	PLC_RECV1.m_nExpId 			:=  PLC_RECV1.m_nExpId 			;      
	PLC_RECV1.m_nAngleStart 	:=	PLC_RECV1.m_nAngleStart 	;   
	PLC_RECV1.m_nAngleEnd  		:=	PLC_RECV1.m_nAngleEnd  		;   
	PLC_RECV1.m_nRotateBegin  	:=  PLC_RECV1.m_nRotateBegin  	; 
	PLC_RECV1.m_nRotateEnd  	:=	PLC_RECV1.m_nRotateEnd  	;   
	PLC_RECV1.m_nKv  			:=	PLC_RECV1.m_nKv  			;       
	PLC_RECV1.m_nMA  			:=	PLC_RECV1.m_nMA  			;        
	PLC_RECV1.m_nMS 			:=	PLC_RECV1.m_nMS 			;        
	PLC_RECV1.m_nFocus 			:=  PLC_RECV1.m_nFocus 			;     
	PLC_RECV1.m_nAcquireFrame 	:=  PLC_RECV1.m_nAcquireFrame 	;
	PLC_RECV1.m_nFramePerCirCle	:=  PLC_RECV1.m_nFramePerCirCle	;
	PLC_RECV1.m_nMoveToward  	:=	PLC_RECV1.m_nMoveToward  	 ;
	PLC_RECV1.m_nServenLamp  	:=  PLC_RECV1.m_nServenLamp  	 ;
	PLC_RECV1.m_nMoveStep  		:=  PLC_RECV1.m_nMoveStep  		 ;  
	PLC_RECV1.m_nPitchValue   	:=  PLC_RECV1.m_nPitchValue   	 ;
	PLC_RECV1.m_nCircleCount  	:=  PLC_RECV1.m_nCircleCount  	 ;
	PLC_RECV1.m_nControlState 	:=  PLC_RECV1.m_nControlState 	 ;
	PLC_RECV1.m_fScanTop 		:=	PLC_RECV1.m_fScanTop 		 ;    
	PLC_RECV1.m_fScanBottom 	:=	PLC_RECV1.m_fScanBottom 	 ;  
	PLC_RECV1.m_fSecondPerCicle	:=  PLC_RECV1.m_fSecondPerCicle	;
	PLC_RECV1.m_nSamplingRate  	:=  PLC_RECV1.m_nSamplingRate  	;
	PLC_RECV1.m_nPrepareState 	:=  PLC_RECV1.m_nPrepareState 	 ;
	PLC_RECV1.m_nScanMoveType	:=	PLC_RECV1.m_nScanMoveType	;  
	PLC_RECV1.m_nCircleIndex 	:=	PLC_RECV1.m_nCircleIndex 	;  
	PLC_RECV1.m_nPLCMaCoeff 	:=	PLC_RECV1.m_nPLCMaCoeff 	 ;  
	PLC_RECV1.m_nLastMsg  		:=  PLC_RECV1.m_nLastMsg  		;    
	PLC_RECV1.m_nDelayTime 		:=  PLC_RECV1.m_nDelayTime 		;       
	PLC_RECV1.yuliu_2			:=	PLC_RECV1.yuliu_2			 ;       
	PLC_RECV1.yuliu_3 			:=  PLC_RECV1.yuliu_3 			 ;      	
END_IF
END_ACTION

ACTION APLC_SENG:

(*---------------------------------PLC发送数据------------------------------------*)//大端发送机制
(*第一部分，发送数据赋值,待补充*)
	IF PLC_RECV1.m_nSocketType=1 THEN
    	PLC_SEND1.m_nSocketType	  := 1;//心跳指令，默认为3，留待判断连接状态。
	ELSE
    	PLC_SEND1.m_nSocketType	  := 3;//心跳指令，默认为3，留待判断连接状态。
	END_IF                                                                            
	PLC_SEND1.m_nCurrentAngle	:= LREAL_TO_REAL(Axis_XZ.XZ_AxisState.rActPosition);//为设备当前的旋转角度，单位为角度制下的单位，为度。数精度为1度；                                                             
	PLC_SEND1.m_nBedHeight		:= Entity_IO.rRealPos+710; //为床高，单位为毫米，数据范围为0 - 2000mm；                                                                 
	PLC_SEND1.m_nBedMovePos		:= LREAL_TO_REAL(Axis_QJ.QJ_AxisState.rActPosition);//为床移动距离，以床与探测板的垂直面交线为起点，单位为毫米，数据范围为0 - 3000mm；//增加了偏移                                                 
//	PLC_SEND1.m_nExpStates		:= 22;//为曝光状态，枚举值，0:idle（空闲） 1:prep（训机） 2: ready（训机结束，准备完成，可以出束） 3: XrayOn（出射线） 4:XrayOff（关射线） 5 error；
	PLC_SEND1.m_nExpCount		:= PLC_PRG.iActNumPulse;//为曝光的次数，对应曝光的图像张数；                                                                              
//	PLC_SEND1.m_nFocus			:= XRAY_RS485.Feedback_nFocus;//焦点大小，0为大焦点 1为小焦点， 焦点具体对应的值由plc设置；        //修改为按键提示                                                      
	PLC_SEND1.m_nMHuValue		:= DT_Xray.Feedback_nMHuValue;//热容量，单位MHu ，实际热容量*100得到，实际热容量为小数；                                                               
	PLC_SEND1.m_nDirectionState	:= BOOL_TO_UDINT(PLC_PRG.bSendQuickCTAngle);                                                                  
//	PLC_SEND1.m_nMoveState		:= 22;//起始、终止状态， 默认值-1， 0为当前扫描方案（与常规意义不同，注意区别）处于准备好状态，可以准备扫描；1为当前扫描方案结束，运动过程中值为-1                      
	PLC_SEND1.m_nError			:= DT_Xray.iAlarmNum;//错误码使用，由王（风杰）工具体阐述内容                                                                            
	PLC_SEND1.m_fSpeed			:= LREAL_TO_REAL(Axis_XZ.XZ_AxisState.rActVelocity);//为设备的旋转速度，单位为度/秒，精度0.01度/秒；                                                                     
	PLC_SEND1.m_fKv				:= DT_Xray.Feedback_Kv;//管电压，单位为kv（千伏），精度0.01；                                                                          
	PLC_SEND1.m_fMA				:= DT_Xray.Feedback_mA;//管电流，单位为mA（毫安），精度0.01；                                                                          
	PLC_SEND1.m_fMs				:= DT_Xray.Feedback_ms;//曝光时间，单位为ms（毫秒），精度0.01；                                                                         
	PLC_SEND1.m_nSamplingRate	:= PLC_RECV1.m_nFramePerCirCle;//采样率，有3个选项：2400帧/圈；1200帧/圈；600帧/圈                                                               
//	PLC_SEND1.m_nScanProType	:= 22;//执行扫描方案的类型，0为自动扫描，1为手动扫描，2为无设置意义的值，默认值为2                                                        
	PLC_SEND1.PLC_State			:= GVL_State.iPLC_State;//PLC状态机状态                                                                                             
	PLC_SEND1.XRAY_State		:= GVL_State.iXray_State;//射线源状态                                                                                     
	PLC_SEND1.AxisErrorID		:= QJ_Error+XZ_Error*65536; //电机错误报警位,各占16位 
    PLC_SEND1.m_nFocusX			:= DT_Xray.Feedback_nFocus;//反馈的焦点

(**处理电机Errstop状态下没有故障吗的情况*)	
	IF Axis_XZ.XZ_AxisState.bAxisErr THEN
		XZ_Error:= Axis_XZ.XZ_AxisState.ErrorID ;
	ELSE
		IF  Axis_XZ.XZ_AxisState.bErrStop THEN
			XZ_Error:= 444 ; 
		ELSE
			XZ_Error:=0;
		END_IF
	END_IF
	
	IF Axis_QJ.QJ_AxisState.bAxisErr THEN
		XZ_Error:= Axis_QJ.QJ_AxisState.ErrorID ;
	ELSE
		IF  Axis_QJ.QJ_AxisState.bErrStop THEN
			QJ_Error:= 444 ; 
		ELSE
			QJ_Error:=0;
		END_IF
	END_IF
	                               
(*第二部分，发送数据发送*)
(*1,//心跳指令，默认为3，留待判断连接状态。*)
	abyWriteData[3]:=UDINT_TO_BYTE(ROR((PLC_SEND1.m_nSocketType AND 16#FF000000),24));
	abyWriteData[2]:=UDINT_TO_BYTE(ROR((PLC_SEND1.m_nSocketType AND 16#FF0000),16));
	abyWriteData[1]:=UDINT_TO_BYTE(ROR((PLC_SEND1.m_nSocketType AND 16#FF00),8));
	abyWriteData[0]:=UDINT_TO_BYTE(PLC_SEND1.m_nSocketType);
	
(*2//为设备当前的旋转角度，单位为角度制下的单位，为度，数精度为1度*)
	RealByte1[0].rData:=PLC_SEND1.m_nCurrentAngle;	
	abyWriteData[4]:=RealByte1[0].wByte[0];
	abyWriteData[5]:=RealByte1[0].wByte[1];
	abyWriteData[6]:=RealByte1[0].wByte[2];
	abyWriteData[7]:=RealByte1[0].wByte[3];
	
(*3//为床高，单位为毫米，数据范围为0 - 2000mm；*)
	RealByte1[1].rData:=PLC_SEND1.m_nBedHeight;	
	abyWriteData[8]:=RealByte1[1].wByte[0];
	abyWriteData[9]:=RealByte1[1].wByte[1];
	abyWriteData[10]:=RealByte1[1].wByte[2];
	abyWriteData[11]:=RealByte1[1].wByte[3];
	
(*4//为床移动距离，以床与探测板的垂直面交线为起点，单位为毫米，数据范围为0 - 3000mm；*)
	RealByte1[2].rData:=PLC_SEND1.m_nBedMovePos;	
	abyWriteData[12]:=RealByte1[2].wByte[0];
	abyWriteData[13]:=RealByte1[2].wByte[1];
	abyWriteData[14]:=RealByte1[2].wByte[2];
	abyWriteData[15]:=RealByte1[2].wByte[3];
	
(*5//为曝光状态，枚举值，0:idle（空闲） 1:prep（训机） 2: ready（训机结束，准备完成，可以出束） 3: XrayOn（出射线） 4:XrayOff（关射线） 5 error；*)
	abyWriteData[19]:=UDINT_TO_BYTE(ROR((PLC_SEND1.m_nExpStates AND 16#FF000000),24));
	abyWriteData[18]:=UDINT_TO_BYTE(ROR((PLC_SEND1.m_nExpStates AND 16#FF0000),16));
	abyWriteData[17]:=UDINT_TO_BYTE(ROR((PLC_SEND1.m_nExpStates AND 16#FF00),8));
	abyWriteData[16]:=UDINT_TO_BYTE(PLC_SEND1.m_nExpStates);
	
(*6//为曝光的次数，对应曝光的图像张数*)
	abyWriteData[23]:=UDINT_TO_BYTE(ROR((PLC_SEND1.m_nExpCount AND 16#FF000000),24));
	abyWriteData[22]:=UDINT_TO_BYTE(ROR((PLC_SEND1.m_nExpCount AND 16#FF0000),16));
	abyWriteData[21]:=UDINT_TO_BYTE(ROR((PLC_SEND1.m_nExpCount AND 16#FF00),8));
	abyWriteData[20]:=UDINT_TO_BYTE(PLC_SEND1.m_nExpCount AND 16#FF);
	
(*7//焦点大小，0为大焦点 1为小焦点， 焦点具体对应的值由plc设置；*)
	abyWriteData[27]:=UDINT_TO_BYTE(ROR((PLC_SEND1.m_nFocus AND 16#FF000000),24));
	abyWriteData[26]:=UDINT_TO_BYTE(ROR((PLC_SEND1.m_nFocus AND 16#FF0000),16));
	abyWriteData[25]:=UDINT_TO_BYTE(ROR((PLC_SEND1.m_nFocus AND 16#FF00),8));
	abyWriteData[24]:=UDINT_TO_BYTE(PLC_SEND1.m_nFocus);

(*8////热容量，单位MHu ，实际热容量*100得到，实际热容量为小数；*)
	RealByte1[3].rData:=PLC_SEND1.m_nMHuValue;	
	abyWriteData[28]:=RealByte1[3].wByte[0];
	abyWriteData[29]:=RealByte1[3].wByte[1];
	abyWriteData[30]:=RealByte1[3].wByte[2];
	abyWriteData[31]:=RealByte1[3].wByte[3];

(*9.;//当前旋转状态，默认值0， 1为正转，2为反转，停止为0*)	
	abyWriteData[35]:=UDINT_TO_BYTE(ROR((PLC_SEND1.m_nDirectionState AND 16#FF000000),24));
	abyWriteData[34]:=UDINT_TO_BYTE(ROR((PLC_SEND1.m_nDirectionState AND 16#FF0000),16));
	abyWriteData[33]:=UDINT_TO_BYTE(ROR((PLC_SEND1.m_nDirectionState AND 16#FF00),8));
	abyWriteData[32]:=UDINT_TO_BYTE(PLC_SEND1.m_nDirectionState);
	
(*10.起始、终止状态， 默认值0， 1为当前扫描方案（与常规意义不同，注意区别）处于准备好状态，可以准备扫描；2为当前扫描方案结束，运动过程中值为0*)
	abyWriteData[39]:=UDINT_TO_BYTE(ROR((PLC_SEND1.m_nMoveState AND 16#FF000000),24));
	abyWriteData[38]:=UDINT_TO_BYTE(ROR((PLC_SEND1.m_nMoveState AND 16#FF0000),16));
	abyWriteData[37]:=UDINT_TO_BYTE(ROR((PLC_SEND1.m_nMoveState AND 16#FF00),8));
	abyWriteData[36]:=UDINT_TO_BYTE(PLC_SEND1.m_nMoveState);
	
(*11.//错误码使用*)
	abyWriteData[43]:=UDINT_TO_BYTE(ROR((PLC_SEND1.m_nError AND 16#FF000000),24));
	abyWriteData[42]:=UDINT_TO_BYTE(ROR((PLC_SEND1.m_nError AND 16#FF0000),16));
	abyWriteData[41]:=UDINT_TO_BYTE(ROR((PLC_SEND1.m_nError AND 16#FF00),8));
	abyWriteData[40]:=UDINT_TO_BYTE(PLC_SEND1.m_nError AND 16#FF);//旋转电机错误码
	
(*12.//为设备的旋转速度，单位为度/秒，精度0.01度/秒；*)
	RealByte1[4].rData:=PLC_SEND1.m_fSpeed;	
	abyWriteData[44]:=RealByte1[4].wByte[0];
	abyWriteData[45]:=RealByte1[4].wByte[1];
	abyWriteData[46]:=RealByte1[4].wByte[2];
	abyWriteData[47]:=RealByte1[4].wByte[3];
	
(*13.//管电压，单位为kv（千伏），精度1；*)
	abyWriteData[51]:=UDINT_TO_BYTE(ROR((PLC_SEND1.m_fKv AND 16#FF000000),24));
	abyWriteData[50]:=UDINT_TO_BYTE(ROR((PLC_SEND1.m_fKv AND 16#FF0000),16));
	abyWriteData[49]:=UDINT_TO_BYTE(ROR((PLC_SEND1.m_fKv AND 16#FF00),8));
	abyWriteData[48]:=UDINT_TO_BYTE(PLC_SEND1.m_fKv AND 16#FF);
	
(*14.//管电流，单位为mA（毫安），精度0.1*)
	RealByte1[6].rData:=PLC_SEND1.m_fMA;	
	abyWriteData[52]:=RealByte1[6].wByte[0];
	abyWriteData[53]:=RealByte1[6].wByte[1];
	abyWriteData[54]:=RealByte1[6].wByte[2];
	abyWriteData[55]:=RealByte1[6].wByte[3];

(*15.//曝光时间，单位为ms（毫秒），精度0.01；*)
	RealByte1[7].rData:=PLC_SEND1.m_fMs;	
	abyWriteData[56]:=RealByte1[7].wByte[0];
	abyWriteData[57]:=RealByte1[7].wByte[1];
	abyWriteData[58]:=RealByte1[7].wByte[2];
	abyWriteData[59]:=RealByte1[7].wByte[3];
	
(*16.//采样率，有3个选项：2400帧/圈；1200帧/圈；600帧/圈*)
	abyWriteData[63]:=UDINT_TO_BYTE(ROR((PLC_SEND1.m_nSamplingRate AND 16#FF000000),24));
	abyWriteData[62]:=UDINT_TO_BYTE(ROR((PLC_SEND1.m_nSamplingRate AND 16#FF0000),16));
	abyWriteData[61]:=UDINT_TO_BYTE(ROR((PLC_SEND1.m_nSamplingRate AND 16#FF00),8));
	abyWriteData[60]:=UDINT_TO_BYTE(PLC_SEND1.m_nSamplingRate AND 16#FF);
	
(*17.//执行扫描方案的类型，0为自动扫描，1为手动扫描，2为无设置意义的值，默认值为2*)
	abyWriteData[67]:=UDINT_TO_BYTE(ROR((PLC_SEND1.m_nScanProType AND 16#FF000000),24));
	abyWriteData[66]:=UDINT_TO_BYTE(ROR((PLC_SEND1.m_nScanProType AND 16#FF0000),16));
	abyWriteData[65]:=UDINT_TO_BYTE(ROR((PLC_SEND1.m_nScanProType AND 16#FF00),8));
	abyWriteData[64]:=UDINT_TO_BYTE(PLC_SEND1.m_nScanProType AND 16#FF);
	
(*18.//PLC工作状态*)
	abyWriteData[71]:=UDINT_TO_BYTE(ROR((PLC_SEND1.PLC_State AND 16#FF000000),24));
	abyWriteData[70]:=UDINT_TO_BYTE(ROR((PLC_SEND1.PLC_State AND 16#FF0000),16));//
	abyWriteData[69]:=UDINT_TO_BYTE(ROR((PLC_SEND1.PLC_State AND 16#FF00),8));	///
	abyWriteData[68]:=UDINT_TO_BYTE(PLC_SEND1.PLC_State AND 16#FF);				//PLC状态机
	
(*19.//XRAY状态*)
	abyWriteData[75]:=UDINT_TO_BYTE(ROR((PLC_SEND1.XRAY_State AND 16#FF000000),24));
	abyWriteData[74]:=UDINT_TO_BYTE(ROR((PLC_SEND1.XRAY_State AND 16#FF0000),16));  
	abyWriteData[73]:=UDINT_TO_BYTE(ROR((PLC_SEND1.XRAY_State AND 16#FF00),8));     
	abyWriteData[72]:=UDINT_TO_BYTE(PLC_SEND1.XRAY_State AND 16#FF);  //射线源状态机              
	
(*20.//电机错误码*)
	abyWriteData[79]:=UDINT_TO_BYTE(ROR((PLC_SEND1.AxisErrorID AND 16#FF000000),24));//旋转电机故障码
	abyWriteData[78]:=UDINT_TO_BYTE(ROR((PLC_SEND1.AxisErrorID AND 16#FF0000),16));//旋转电机故障码
	abyWriteData[77]:=UDINT_TO_BYTE(ROR((PLC_SEND1.AxisErrorID AND 16#FF00),8));//前进电机故障码
	abyWriteData[76]:=UDINT_TO_BYTE(PLC_SEND1.AxisErrorID AND 16#FF);//前进电机故障码
	
(*21.射线源大小焦点反馈*)
	abyWriteData[83]:=UDINT_TO_BYTE(ROR((PLC_SEND1.m_nFocusX AND 16#FF000000),24));//
	abyWriteData[82]:=UDINT_TO_BYTE(ROR((PLC_SEND1.m_nFocusX AND 16#FF0000),16));//
	abyWriteData[81]:=UDINT_TO_BYTE(ROR((PLC_SEND1.m_nFocusX AND 16#FF00),8));//
	abyWriteData[80]:=UDINT_TO_BYTE(PLC_SEND1.m_nFocusX AND 16#FF);//反馈焦点
	
	
(*	TEST
	PLC_SEND1.m_nSocketType	  	:= 1;//心跳指令，默认为3，留待判断连接状态。                                                                            
	PLC_SEND1.m_nCurrentAngle	:= 2.1;//为设备当前的旋转角度，单位为角度制下的单位，为度。数精度为1度；                                                               
	PLC_SEND1.m_nBedHeight		:= 3.2;//为床高，单位为毫米，数据范围为0 - 2000mm；                                                                  
	PLC_SEND1.m_nBedMovePos		:= 4.3;//为床移动距离，以床与探测板的垂直面交线为起点，单位为毫米，数据范围为0 - 3000mm；                                                  
	PLC_SEND1.m_nExpStates		:= 5;//为曝光状态，枚举值，0:idle（空闲） 1:prep（训机） 2: ready（训机结束，准备完成，可以出束） 3: XrayOn（出射线） 4:XrayOff（关射线） 5 error；
	PLC_SEND1.m_nExpCount		:= 6;//为曝光的次数，对应曝光的图像张数；                                                                              
	PLC_SEND1.m_nFocus			:= 7;//焦点大小，0为大焦点 1为小焦点， 焦点具体对应的值由plc设置；                                                              
	PLC_SEND1.m_nMHuValue		:= 8.1;//热容量，单位MHu ，实际热容量*100得到，实际热容量为小数；                                                               
	PLC_SEND1.m_nDirectionState	:= 9;//当前旋转状态，默认值-1， 0为正转，1为反转，停止为-1                                                                  
	PLC_SEND1.m_nMoveState		:= 10;//起始、终止状态， 默认值-1， 0为当前扫描方案（与常规意义不同，注意区别）处于准备好状态，可以准备扫描；1为当前扫描方案结束，运动过程中值为-1                      
	PLC_SEND1.m_nError			:= 11;//错误码使用，由王（风杰）工具体阐述内容                                                                            
	PLC_SEND1.m_fSpeed			:= 12.2;//为设备的旋转速度，单位为度/秒，精度0.01度/秒；                                                                     
	PLC_SEND1.m_fKv				:= 13;//管电压，单位为kv（千伏），精度0.01；                                                                          
	PLC_SEND1.m_fMA				:= 14.3;//管电流，单位为mA（毫安），精度0.01；                                                                          
	PLC_SEND1.m_fMs				:= 15.3;//曝光时间，单位为ms（毫秒），精度0.01；                                                                         
	PLC_SEND1.m_nSamplingRate	:= 16;//采样率，有3个选项：2400帧/圈；1200帧/圈；600帧/圈                                                               
	PLC_SEND1.m_nScanProType	:= 17;//执行扫描方案的类型，0为自动扫描，1为手动扫描，2为无设置意义的值，默认值为2                                                        
	PLC_SEND1.PLC_State			:= GVL_State.iPLC_State;//PLC状态机状态                                                                                             
	PLC_SEND1.XRAY_State		:= 18;//电机错误报警位,各占16位                                                                                             
	PLC_SEND1.AxisErrorID		:= Axis_QJ.QJ_AxisState.ErrorID+Axis_XZ.XZ_AxisState.ErrorID*65536;//一共20个数据 
*)
END_ACTION

END_PROGRAM

// Device/Application/PLC_PRG

PROGRAM PLC_PRG
VAR
	//(bHomingDone AND XRAY_RS485.Main_Step=20) OR Entity_IO.bEmergencyStop
	count: BYTE;
	bOver: BOOL; //关机结束指令
	bSelfOK: BOOL;//自检成功标志
	bDebug_Laser:BOOL;
	TOF_Laser	:TOF;//激光灯控制
	TP_Laser	:Standard.TP;
	F_TRIG1		:Standard.F_TRIG;//激光灯按钮关闭
	R_TRIG1		:Standard.R_TRIG;//激光灯按钮关闭
	TOF_ET:TIME;
	TOF_PowerDelay,TOF_PowerDelayMax: Standard.TOF;//延迟断电继电器控制
	LS_GetIPAddress_1: LS_GetIPAddress;
	LS_SetIPAddress_1: LS_SetIPAddress;
	rPLC_Load:REAL;
	LS_SetDintDT_1:LS_SysLib.LS_SetDintDT;
	bSetSysTime:BOOL;
	LS_ReadDintDT_1:LS_SysLib.LS_ReadDintDT;
	
	TON_StopScan:Standard.TON;

	iValidTrigger:UINT;
	iHopeNumPulse:UINT:=108;
	
	Step_Home,Step_Idle:INT;//待机模式下工作步骤
	Step_StaticDR,Step_DynamicDR:INT;//静态DR和动态DR
	Step_StandardCT,Step_Scout,Step_CBCT,Step_QuickCT:INT;//静态CT
	Step_Air_High,Step_Air_Quick,Step_Air:INT;//空气校正流程
	Step_ShutDown:INT;
	bStaticDRLast,bStandardCTLast,bScoutLast,bCBCTLast,bQuickCTLast:BOOL;//最后一次扫描标志位
	bAirLast1,bAirLast2,bAirLast3:BOOL;//空气校正下的最后一次标志位
	TimeScoutExp:TIME;//定位像曝光时间
	TimeDRExpS,TimeDRExpD:TIME;//静态和动态DR曝光时间
	bCBCT_AUTO_Manual:BOOL;//自动扫还是手动扫标志位
	bPulseOneStop:BOOL;//回到待机模式下立刻停止
	
	iSamplingRate:UINT;//CBCT采样率
	iHopePulse:UINT;//
	EncoderNum1:DINT;//编码器数值
	iStartTrigger1:DINT;//开始扫数值
	DB_EncoderNum1:DINT;
	iActNumPulse:UINT;//有效触发次数
	i: INT;
	
	TON_CT_J:ARRAY[1..50] OF Standard.TON;//静态模式下TON
	TON_CT_G:ARRAY[1..50] OF Standard.TON;//标准高清快速模式下TON
	TON_DR_S:ARRAY[1..50] OF Standard.TON;//标准高清快速模式下TON
	TON_Air:ARRAY[1..50] OF Standard.TON;//空气校正模式下的TON
	
	bXaryTwo_TEMP:BOOL; //二档输出中间变量
	
	TON_I00,TON_I10,TON_I20,TON_I30,TON_I40,TON_I50:Standard.TON;

	R_DR_Jump,R_CT_J1,R_CT_J,R_TRIG_G1,R_TRIG_G2,R_TRIG_C220,R_TRIG_Jog,R_TRIG_Jog1,R_TRIG_Jog2,R_MoveRecordPos,R_RelStop,R_Static_Tigger:Standard.R_TRIG;
	F_DR_Jump,F_TRIG_G1,F_TRIG_G2,F_TRIG_Jog,F_TRIG_Jog1,F_TRIG_Jog2,F_TRIG_S,F_TRIG_S1:Standard.F_TRIG;//
	
	TOF_DR111:TOF;
	HandSelfStep: INT;
	bErrorReset:BOOL;
	bHomingDone: BOOL;
	
	bGetPLC_IP,bSetPLC_IP,bGetPLC_Load:BOOL;
	
	XZ_Velocity:REAL:=10;//设置不扫描时快速到扫描位的速度
	TON_Home:TON;
	TON_Error,TON_Error1,TON_Power,TON_Home1,TON_IDLE,CTBOX_TON1,TON_Wait:Standard.TON;
	TOF_JOG,TOF_DR22,CTBOX_TOF1:Standard.TOF;
	
	R_TRIG_debug,R_TRIG_debug2:Standard.R_TRIG;
	aaa,bbb,ccc,ddd:BOOL;
	bXrayOneDR:BOOL;
	Blink_Air1,Blink_Air2:BLINK;
	iTriggerNum1,iTriggerNum2:INT;
	R_Trig_Air1,R_Trig_Air2:Standard.R_TRIG;
	F_Trig_Air1,F_Trig_Air2:Standard.R_TRIG;
	bAirHigh:BOOL;
	
	Blink_StaticDR_Temp:Blink;//测试DR
	
	DelayTime,ExpTimeQuick:TIME;
	Minute1,Minute2:UINT;
	Second1,Second2:UINT;
	R_TRIG_SS:Standard.R_TRIG;
	F_TRIG_SS:Standard.F_TRIG;
	
	bSetXZ_Zero:BOOL;
	rSetXZ_Zero:REAL;
	
	bSendQuickCTAngle:BOOL;
	iAngleStartQuickCT:REAL;

	bTestFLU:BOOL;
END_VAR

VAR_OUTPUT	
	LampCmd5,LampCmd6,LampCmd7,LampCmd8:E_LampCmd;
END_VAR

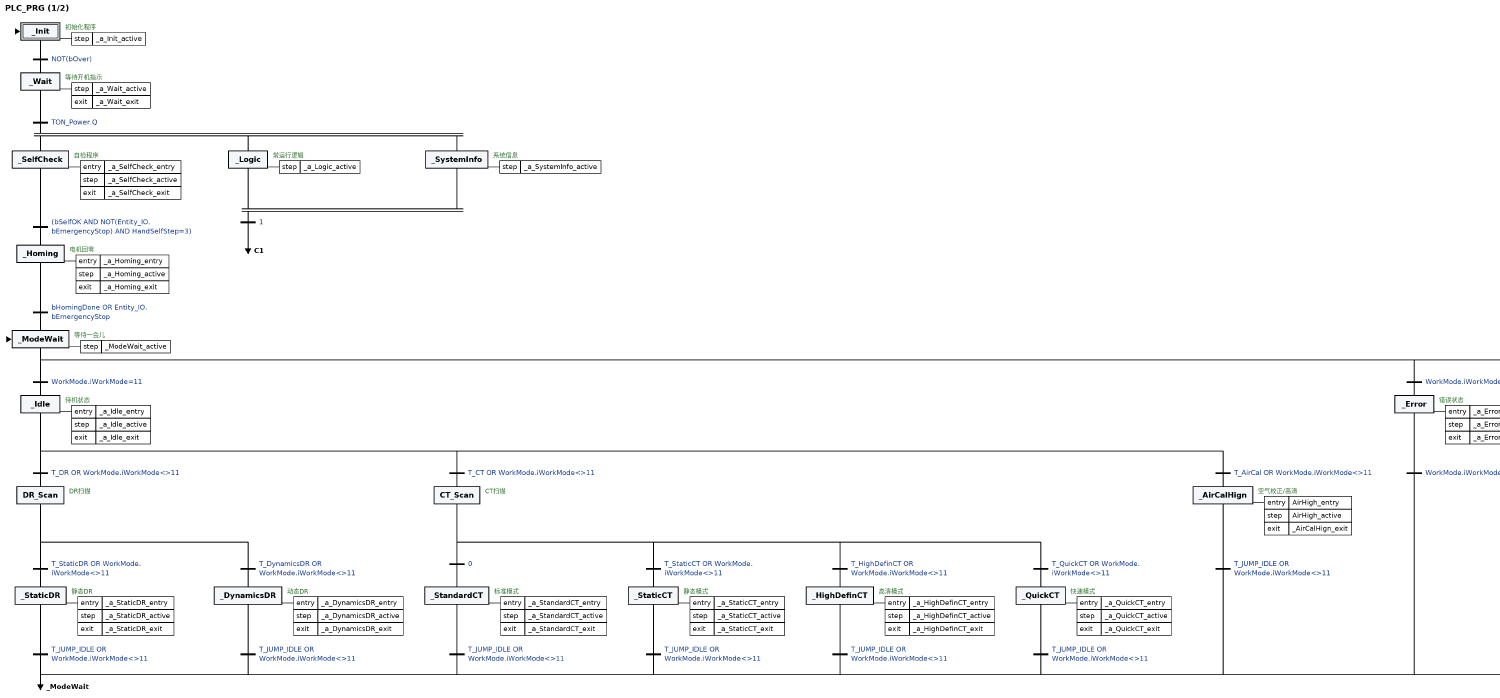
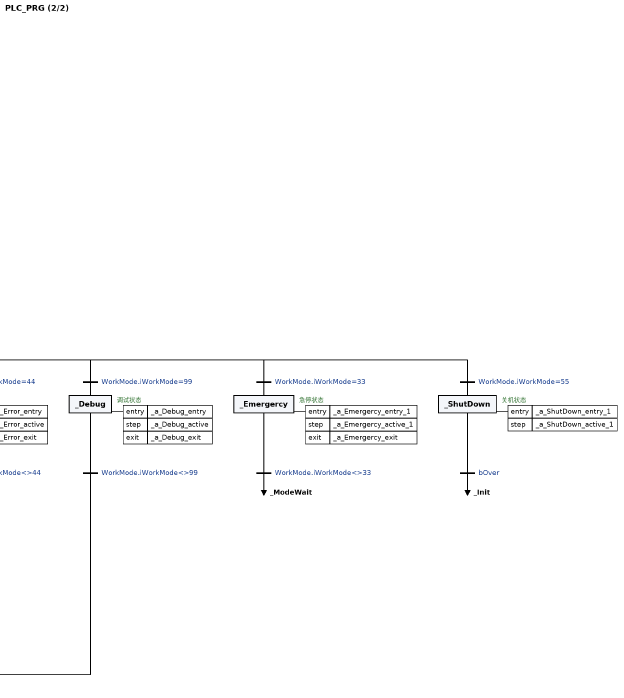
// 初始化程序
INITIAL_STEP _Init:
    _a_Init_active(N);  // step action
END_STEP
TRANSITION FROM _Init TO _Wait
    := NOT(bOver);
END_TRANSITION
// 等待开机指示
STEP _Wait:
    _a_Wait_active(N);  // step action
    _a_Wait_exit(P0);  // exit action
END_STEP
TRANSITION FROM _Wait TO (_SelfCheck, _Logic, _SystemInfo)
    := TON_Power.Q;
END_TRANSITION
// 自检程序
STEP _SelfCheck:
    _a_SelfCheck_entry(P1);  // entry action
    _a_SelfCheck_active(N);  // step action
    _a_SelfCheck_exit(P0);  // exit action
END_STEP
TRANSITION FROM _SelfCheck TO _Homing
    := (bSelfOK AND NOT(Entity_IO.bEmergencyStop) AND HandSelfStep=3);
END_TRANSITION
// 电机回零
STEP _Homing:
    _a_Homing_entry(P1);  // entry action
    _a_Homing_active(N);  // step action
    _a_Homing_exit(P0);  // exit action
END_STEP
TRANSITION FROM _Homing TO _ModeWait
    := bHomingDone OR Entity_IO.bEmergencyStop;
END_TRANSITION
// 等待一会儿
STEP _ModeWait:
    _ModeWait_active(N);  // step action
END_STEP
TRANSITION FROM _ModeWait TO _Idle
    := WorkMode.iWorkMode=11;
END_TRANSITION
// 待机状态
STEP _Idle:
    _a_Idle_entry(P1);  // entry action
    _a_Idle_active(N);  // step action
    _a_Idle_exit(P0);  // exit action
END_STEP
TRANSITION FROM _Idle TO DR_Scan
    := T_DR OR WorkMode.iWorkMode<>11;
END_TRANSITION
// DR扫描
STEP DR_Scan:
END_STEP
TRANSITION FROM DR_Scan TO _StaticDR
    := T_StaticDR OR WorkMode.iWorkMode<>11;
END_TRANSITION
// 静态DR
STEP _StaticDR:
    _a_StaticDR_entry(P1);  // entry action
    _a_StaticDR_active(N);  // step action
    _a_StaticDR_exit(P0);  // exit action
END_STEP
TRANSITION FROM _StaticDR TO _ModeWait
    := T_JUMP_IDLE OR WorkMode.iWorkMode<>11;
END_TRANSITION
TRANSITION FROM DR_Scan TO _DynamicsDR
    := T_DynamicsDR OR WorkMode.iWorkMode<>11;
END_TRANSITION
// 动态DR
STEP _DynamicsDR:
    _a_DynamicsDR_entry(P1);  // entry action
    _a_DynamicsDR_active(N);  // step action
    _a_DynamicsDR_exit(P0);  // exit action
END_STEP
TRANSITION FROM _DynamicsDR TO _ModeWait
    := T_JUMP_IDLE OR WorkMode.iWorkMode<>11;
END_TRANSITION
TRANSITION FROM _Idle TO CT_Scan
    := T_CT OR WorkMode.iWorkMode<>11;
END_TRANSITION
// CT扫描
STEP CT_Scan:
END_STEP
TRANSITION FROM CT_Scan TO _StandardCT
    := 0;
END_TRANSITION
// 标准模式
STEP _StandardCT:
    _a_StandardCT_entry(P1);  // entry action
    _a_StandardCT_active(N);  // step action
    _a_StandardCT_exit(P0);  // exit action
END_STEP
TRANSITION FROM _StandardCT TO _ModeWait
    := T_JUMP_IDLE OR WorkMode.iWorkMode<>11;
END_TRANSITION
TRANSITION FROM CT_Scan TO _StaticCT
    := T_StaticCT OR WorkMode.iWorkMode<>11;
END_TRANSITION
// 静态模式
STEP _StaticCT:
    _a_StaticCT_entry(P1);  // entry action
    _a_StaticCT_active(N);  // step action
    _a_StaticCT_exit(P0);  // exit action
END_STEP
TRANSITION FROM _StaticCT TO _ModeWait
    := T_JUMP_IDLE OR WorkMode.iWorkMode<>11;
END_TRANSITION
TRANSITION FROM CT_Scan TO _HighDefinCT
    := T_HighDefinCT OR WorkMode.iWorkMode<>11;
END_TRANSITION
// 高清模式
STEP _HighDefinCT:
    _a_HighDefinCT_entry(P1);  // entry action
    _a_HighDefinCT_active(N);  // step action
    _a_HighDefinCT_exit(P0);  // exit action
END_STEP
TRANSITION FROM _HighDefinCT TO _ModeWait
    := T_JUMP_IDLE OR WorkMode.iWorkMode<>11;
END_TRANSITION
TRANSITION FROM CT_Scan TO _QuickCT
    := T_QuickCT OR WorkMode.iWorkMode<>11;
END_TRANSITION
// 快速模式
STEP _QuickCT:
    _a_QuickCT_entry(P1);  // entry action
    _a_QuickCT_active(N);  // step action
    _a_QuickCT_exit(P0);  // exit action
END_STEP
TRANSITION FROM _QuickCT TO _ModeWait
    := T_JUMP_IDLE OR WorkMode.iWorkMode<>11;
END_TRANSITION
TRANSITION FROM _Idle TO _AirCalHign
    := T_AirCal OR WorkMode.iWorkMode<>11;
END_TRANSITION
// 空气校正/高清
STEP _AirCalHign:
    AirHigh_entry(P1);  // entry action
    AirHigh_active(N);  // step action
    _AirCalHign_exit(P0);  // exit action
END_STEP
TRANSITION FROM _AirCalHign TO _ModeWait
    := T_JUMP_IDLE OR WorkMode.iWorkMode<>11;
END_TRANSITION
TRANSITION FROM _ModeWait TO _Error
    := WorkMode.iWorkMode=44;
END_TRANSITION
// 错误状态
STEP _Error:
    _a_Error_entry(P1);  // entry action
    _a_Error_active(N);  // step action
    _a_Error_exit(P0);  // exit action
END_STEP
TRANSITION FROM _Error TO _ModeWait
    := WorkMode.iWorkMode<>44;
END_TRANSITION
TRANSITION FROM _ModeWait TO _Debug
    := WorkMode.iWorkMode=99;
END_TRANSITION
// 调试状态
STEP _Debug:
    _a_Debug_entry(P1);  // entry action
    _a_Debug_active(N);  // step action
    _a_Debug_exit(P0);  // exit action
END_STEP
TRANSITION FROM _Debug TO _ModeWait
    := WorkMode.iWorkMode<>99;
END_TRANSITION
TRANSITION FROM _ModeWait TO _Emergercy
    := WorkMode.iWorkMode=33;
END_TRANSITION
// 急停状态
STEP _Emergercy:
    _a_Emergercy_entry_1(P1);  // entry action
    _a_Emergercy_active_1(N);  // step action
    _a_Emergercy_exit(P0);  // exit action
END_STEP
TRANSITION FROM _Emergercy TO _ModeWait
    := WorkMode.iWorkMode<>33;
END_TRANSITION
TRANSITION FROM _ModeWait TO _ShutDown
    := WorkMode.iWorkMode=55;
END_TRANSITION
// 关机状态
STEP _ShutDown:
    _a_ShutDown_entry_1(P1);  // entry action
    _a_ShutDown_active_1(N);  // step action
END_STEP
TRANSITION FROM _ShutDown TO _Init
    := bOver;
END_TRANSITION
// 常运行逻辑
STEP _Logic:
    _a_Logic_active(N);  // step action
END_STEP
// 系统信息
STEP _SystemInfo:
    _a_SystemInfo_active(N);  // step action
END_STEP
TRANSITION FROM (_Logic, _SystemInfo) TO (_Logic, _SystemInfo)
    := 1;
END_TRANSITION
// branch label C1
// branch label B1

ACTION _a_SelfCheck_active:

GVL_State.iPLC_State:=20;

(*目前只检查电机错误*)
	bSelfOK:=NOT(Axis_QJ.QJ_AxisState.bAxisErr OR Axis_XZ.XZ_AxisState.bAxisErr);

(*有错误自动复位*)	
	IF Entity_IO.bEmergencyStop = FALSE  THEN  //急停未被拍下
		CASE HandSelfStep OF
			0:
				IF Axis_QJ.QJ_AxisState.bAxisErr THEN
					Axis_QJ.QJ_AxisCmd.bReset:=TRUE;
				ELSE
					HandSelfStep:=1;
				END_IF
				
			1:
				IF Axis_XZ.XZ_AxisState.bAxisErr THEN
					Axis_XZ.XZ_AxisCmd.bReset:=TRUE;
				ELSE
					HandSelfStep:=2;
				END_IF
				
			2:
				Axis_XZ.XZ_AxisCmd.bReset:=FALSE;
				Axis_QJ.QJ_AxisCmd.bReset:=FALSE;
				HandSelfStep:=3;
				
			3:
				;	
		END_CASE
	END_IF;

(*旋转电机写入电机回零默认参数*)
//	Axis_XZ.XZ_AxisCmd.AxisPara.rHomeAcc:=5.0;
//	Axis_XZ.XZ_AxisCmd.AxisPara.iHomeMode:=10;
//	Axis_XZ.XZ_AxisCmd.AxisPara.rHomeHighSpeed:=10;
//	Axis_XZ.XZ_AxisCmd.AxisPara.rHomeLowSpeed:=5;
	
(*前进写入电机回零默认参数*)
//	Axis_QJ.QJ_AxisCmd.AxisPara.rHomeAcc:=5.0;
//	Axis_QJ.QJ_AxisCmd.AxisPara.iHomeMode:=10;
//	Axis_QJ.QJ_AxisCmd.AxisPara.rHomeHighSpeed:=10;
//	Axis_QJ.QJ_AxisCmd.AxisPara.rHomeLowSpeed:=5;
END_ACTION

ACTION _a_StandardCT_active:

	CASE Step_StandardCT OF 
		0:	//初始化准备流程
			(*1.给上位机发送的数据*)
			WorkStation_TCP.PLC_SEND1.m_nMoveState:=0;			//send[9] //0-准备过程中 1-准备完成 2-曝光中 3-本次扫描结束 
			bStandardCTLast		:=FALSE;
			
			(*2.运动准备数据*)
			(*2.1 写入旋转速度参数*)
			IF WorkStation_TCP.PLC_RECV1.m_fSecondPerCicle<>0 THEN//避免除零
				Axis_XZ.XZ_AxisCmd.AxisPara.rAbsVelocity:=(LIMIT(360/300 ,360/WorkStation_TCP.PLC_RECV1.m_fSecondPerCicle ,360/8));
				XZ_Velocity:=LIMIT(360/300 ,360/(WorkStation_TCP.PLC_RECV1.m_fSecondPerCicle) ,360/8);
			ELSE
				Axis_XZ.XZ_AxisCmd.AxisPara.rAbsVelocity:=8;
			END_IF;
			
			(*3.中间变量复位*)
			FOR i:=1 TO 50 BY 1 DO 
				TON_CT_G[i](IN:= FALSE);
			END_FOR
			Axis_XZ.XZ_AxisCmd.bAbs		:=FALSE;
			Axis_QJ.QJ_AxisCmd.bAbs		:=FALSE;
			Step_StandardCT:=10;
				
		10://按5键，移动床到预设位置，松开即停，机架直接到预设位置
			(*1.发送给上位机的数据*)
			WorkStation_TCP.PLC_SEND1.m_nExpStates	:=1;		//0-准备过程中 1-准备完成 2-曝光中 3-本次扫描结束	
			WorkStation_TCP.PLC_SEND1.m_nMoveState	:=0;		//起始、终止状态， 默认值0， 1为当前扫描方案处于准备好状态，可以准备扫描；2为当前扫描方案结束，运动过程中值为0
			WorkStation_TCP.PLC_SEND1.m_nScanProType:=2;	//扫描方案类型 , 1-手动，0-自动. 
			
			(*2.旋转轴直接运动到目标位置*)
			Axis_XZ.XZ_AxisCmd.AxisPara.rAbsPosition	:=LIMIT(-3,WorkStation_TCP.PLC_RECV1.m_nRotateBegin,363);
			Axis_XZ.XZ_AxisCmd.AxisPara.rAbsVelocity	:=18;
			TON_CT_G[1](IN:=TRUE , PT:=T#500MS);
			Axis_XZ.XZ_AxisCmd.bAbs						:=TON_CT_G[1].Q;
			
			(*3.前进轴运动*)
			R_TRIG_G1(CLK:= CTBOX_RS232.CTBOX_KEY_MoveDistance, Q=> );//触发运动
			F_TRIG_G1(CLK:= CTBOX_RS232.CTBOX_KEY_MoveDistance, Q=> );//触发停止
			
			Axis_QJ.QJ_AxisCmd.bAbs	:=R_TRIG_G1.Q;
			Axis_QJ.QJ_AxisCmd.AxisPara.rAbsPosition	:=LIMIT(0,WorkStation_TCP.PLC_RECV1.m_fScanTop,900);
			Axis_QJ.QJ_AxisCmd.bStop:=F_TRIG_G1.Q;
			
			(*4.5灯逻辑处理*)
			IF ABS(Axis_QJ.QJ_AxisState.rActPosition-WorkStation_TCP.PLC_RECV1.m_fScanTop)>1 THEN
				LampCmd5:=E_LampCmd.慢闪;
				WorkStation_TCP.PLC_SEND1.m_nFocus:=5;			//按键提示0228
			ELSE
				LampCmd5:=E_LampCmd.关闭;
				WorkStation_TCP.PLC_SEND1.m_nFocus:=0;			//关闭按键提示0228
			END_IF
			
			(*5.跳转*)
			TON_CT_G[2](IN:=ABS(Axis_QJ.QJ_AxisState.rActPosition-WorkStation_TCP.PLC_RECV1.m_fScanTop)<1 
				AND ABS(Axis_XZ.XZ_AxisState.rActPosition-WorkStation_TCP.PLC_RECV1.m_nRotateBegin)<1 
				AND Axis_XZ.XZ_AxisState.bStandStill AND Axis_QJ.QJ_AxisState.bStandStill, PT:=T#100MS);
			IF TON_CT_G[2].Q THEN  
				Step_StandardCT:=20;
			END_IF
			
		20:	//射线源参数写入成功标志
			(*1.变量复位*)
			LampCmd5:=E_LampCmd.关闭;
			Axis_XZ.XZ_AxisCmd.bAbs		:=FALSE;
			Axis_QJ.QJ_AxisCmd.bAbs		:=FALSE;
			Axis_QJ.QJ_AxisCmd.bStop	:=FALSE;
			
			(*2.射线源参数写入正常完毕*)
			IF DT_Xray.ExpPara_Step=66 THEN
				Step_StandardCT:=30;
			END_IF
			
		30:	//7灯和8灯开始慢闪
			(*1.给上位机发送的数*)
			WorkStation_TCP.PLC_SEND1.m_nMoveState	:=1;		//起始、终止状态， 默认值0， 1为当前扫描方案处于准备好状态
			WorkStation_TCP.PLC_SEND1.m_nFocus		:=8;		//按键提示0228
			
			(*2.CTBOX灯的状态*)
			LampCmd7:=E_LampCmd.慢闪;
			LampCmd8:=E_LampCmd.慢闪;
			
			TON_CT_G[3](IN:=TRUE , PT:=T#600MS);
			IF TON_CT_G[3].Q THEN
				Step_StandardCT:=40;
			END_IF
		
		40://用户选择自动扫描或手动扫描
			IF CTBOX_RS232.CTBOX_KEY_Auto=FALSE AND CTBOX_RS232.CTBOX_KEY_Manual THEN
				WorkStation_TCP.PLC_SEND1.m_nScanProType:=1;								//扫描方案类型 , 1-手动，0-自动. 
				bCBCT_AUTO_Manual:=TRUE;
			ELSIF CTBOX_RS232.CTBOX_KEY_Auto AND CTBOX_RS232.CTBOX_KEY_Manual=FALSE THEN
				WorkStation_TCP.PLC_SEND1.m_nScanProType:=0;								//扫描方案类型 , 1-手动，0-自动. 
				bCBCT_AUTO_Manual:=FALSE;
			ELSIF CTBOX_RS232.CTBOX_KEY_Auto=FALSE AND CTBOX_RS232.CTBOX_KEY_Manual=FALSE THEN
				;
			ELSIF CTBOX_RS232.CTBOX_KEY_Auto AND CTBOX_RS232.CTBOX_KEY_Manual THEN
				;
			END_IF
			
			IF (CTBOX_RS232.CTBOX_KEY_Auto AND CTBOX_RS232.CTBOX_KEY_Manual=FALSE) OR CTBOX_RS232.CTBOX_KEY_Manual AND CTBOX_RS232.CTBOX_KEY_Auto=FALSE THEN
				Step_StandardCT:=50;
			END_IF
			
		50://7和8灯关闭 
			(*1.给上位机发送的数据*)
			WorkStation_TCP.PLC_SEND1.m_nFocus:=0;	//关闭按键提示0228
			
			(*2.CTBOX灯关闭*)
			LampCmd7:=E_LampCmd.关闭;
			LampCmd8:=E_LampCmd.关闭;
			
			(*3.获取当前编码器数值*)
			iStartTrigger1:=Entity_IO.iEncoderPulse;//只赋值一次
			
			(*4.跳转*)
			TON_CT_G[4](IN:= TRUE, PT:=T#1S);
			IF TON_CT_G[4].Q THEN
				Step_StandardCT:=60;
			END_IF
			
		60://扫描中间态，给跳转用的
			(*1.变量复位*)
			FOR i:=1 TO 50 BY 1 DO 
				TON_CT_G[i](IN:= FALSE);
			END_FOR
			Axis_QJ.QJ_AxisCmd.bAbs:=FALSE;//复位前进轴
			Axis_XZ.XZ_AxisCmd.bAbs:=FALSE;//复位旋转轴
			iActNumPulse:=0;
			Step_StandardCT:=70;
			
		70:
			(*1.发送给上位机的数据*)
			WorkStation_TCP.PLC_SEND1.m_nMoveState	:=1;	//send[9]
			WorkStation_TCP.PLC_SEND1.m_nScanProType:=2;	//send[16]
			
			(*2.射线源参数写入成功，开启透视*)
			IF DT_Xray.ExpPara_Step=66 THEN  //保证写入参数
				Entity_IO.bXaryOne:=TRUE;//开启一二档
				Entity_IO.bXaryTwo:=TRUE;//开启一二档
			END_IF;
			
			(*3.判断是否最后一次扫描*)
			IF WorkStation_TCP.PLC_RECV1.m_nLastMsg=1 THEN
				bStandardCTLast := TRUE;
			ELSE
				bStandardCTLast := FALSE;
			END_IF
			
			(*4.获取上位机发送的采样率,有可能是半扫*)//
			iSamplingRate:=REAL_TO_UINT(UDINT_TO_REAL(WorkStation_TCP.PLC_RECV1.m_nSamplingRate)*ABS(WorkStation_TCP.PLC_RECV1.m_nAngleStart-WorkStation_TCP.PLC_RECV1.m_nAngleEnd)/360);//采样率，有4个选项：2400帧/圈；1200帧/圈；600帧/圈,360帧/圈
			
			(*5.处理多少个脉冲输出一个trigger*)
			CASE iSamplingRate OF 
				360:iHopePulse:=360;
				600:iHopePulse:=216;
				1200:iHopePulse:=108;
				2400:iHopePulse:=54;
				ELSE iHopePulse:=360;
			END_CASE

			(*6.跳转指令*)
			TON_CT_G[5](IN:=TRUE,PT:=T#600MS);
			IF TON_CT_G[5].Q AND Entity_IO.bXaryOne AND Entity_IO.bXaryTwo THEN
				Step_StandardCT:=80;
			END_IF
			
			(*7.计数复位*)
			iActNumPulse:=0;
			
		74:
			Entity_IO.bXaryOne:=FALSE;
			Entity_IO.bXaryTwo:=FALSE;
			GVL_SCAN.bJumpScan:=TRUE;		//结束扫描，射线源超时报警了，EL019，结束扫描
			Step_StandardCT:=74;
			
		80://第一次自动扫描
			(*1.给上位机发送的数*)
			WorkStation_TCP.PLC_SEND1.m_nMoveState	:=2;
			WorkStation_TCP.PLC_SEND1.m_nScanProType:=2;

			(*2.触发旋转轴运动*)
			Axis_XZ.XZ_AxisCmd.AxisPara.rAbsPosition:=LIMIT(-3,WorkStation_TCP.PLC_RECV1.m_nRotateEnd,363);
			Axis_XZ.XZ_AxisCmd.AxisPara.rAbsVelocity:=XZ_Velocity;
			TON_CT_G[6](IN:=TRUE , PT:=T#200MS );
			Axis_XZ.XZ_AxisCmd.bAbs:=TON_CT_G[6].Q;
					
			(*4.开启允许采图指令*)
			(*4.1.获取旋转编码器的数值*)
			EncoderNum1:=Entity_IO.iEncoderPulse;
			(*4.2处理相对脉冲来作为触发*)
			DB_EncoderNum1:=ABS(EncoderNum1-iStartTrigger1);
			iValidTrigger:=DINT_TO_UINT(DB_EncoderNum1 MOD iHopePulse);
			
			IF (iActNumPulse)<=(iSamplingRate+3) THEN			//多加一个1
				IF (iValidTrigger)<=5*iHopePulse / 10 THEN  	//1/3的占空比，这个时间要和上位机下发的扫描时间对应
					Entity_IO.bTriggerOut:=TRUE;
				ELSE
					Entity_IO.bTriggerOut:=FALSE;
				END_IF
			ELSE
				Entity_IO.bTriggerOut:=FALSE;
			END_IF;
			
			(*4.3 计数器计算*)
			F_TRIG_G2(CLK:=Entity_IO.bTriggerOut , Q=>);
			IF F_TRIG_G2.Q THEN iActNumPulse:=iActNumPulse+1;END_IF;

			(*5.跳转,到达终止角度*)
			TON_CT_G[7](IN:= ABS(Axis_XZ.XZ_AxisState.rActPosition-WorkStation_TCP.PLC_RECV1.m_nRotateEnd)<1 AND Axis_XZ.XZ_AxisState.bStandStill, PT:=T#200MS , Q=> , ET=> );	
			IF TON_CT_G[7].Q THEN
				Step_StandardCT:=90;
			END_IF
			
			(*6.一二档信号超时报警，射线源30秒连续开启曝光会报警*)
			TON_CT_G[8](IN:=Entity_IO.bXaryTwo , PT:=T#30S , Q=> , ET=> );
			IF TON_CT_G[8].Q THEN
				Step_StandardCT:=74;	
			END_IF
			
		90://出射线状态结束，采集射线源状态机信息
			(*1.关闭透视信号*)
			Entity_IO.bXaryOne		:=FALSE;
			Entity_IO.bXaryTwo		:=FALSE;
			Axis_XZ.XZ_AxisCmd.bAbs	:=FALSE;
			(*2.跳转*)
			
			IF GVL_State.iXray_State=40 THEN	//DT射线源增加状态 ,回到待机状态 
				Step_StandardCT:=100;
			END_IF
			
		100://中间变量清零1070
			(*1.给上位机发送的数据*)
			WorkStation_TCP.PLC_SEND1.m_nMoveState:=3; //send [9]
			
			(*2.判断是否最后一次扫描*)
			TON_CT_G[9](IN:=TRUE , PT:=T#1S , Q=> , ET=> );
			IF TON_CT_G[9].Q THEN
				IF (WorkStation_TCP.PLC_RECV1.m_nCircleIndex+1)>=(WorkStation_TCP.PLC_RECV1.m_nCircleCount) AND bStandardCTLast THEN //最后一次扫描退出
					GVL_SCAN.bJumpScan:=TRUE;
				END_IF
			END_IF
		
			(*3.不是最后一次增加跳转判断增加跳转接着扫*)
			IF WorkStation_TCP.PLC_RECV1.m_nSocketType=1 THEN 	//增加第二次运动判断，m_nSocketType=1 
				Step_StandardCT:=110;
			END_IF
			
		110://CBCT下的自动扫还是手动扫，根据上位机命令
			IF WorkStation_TCP.PLC_RECV1.m_nScanMoveType=1 THEN
				Step_StandardCT:=200;		//手动扫描
			ELSE
				Step_StandardCT:=120;		//自动扫描
			END_IF
		 
		120://开启自动扫描
			(*1.前进轴自动运动*)
			TON_CT_G[10](IN:=TRUE , PT:=T#300MS , Q=> , ET=> );
			Axis_QJ.QJ_AxisCmd.AxisPara.rAbsPosition:=LIMIT(0,WorkStation_TCP.PLC_RECV1.m_fScanTop,900);
			Axis_QJ.QJ_AxisCmd.bAbs:=TON_CT_G[10].Q;
			
			(*2.给上位机发送的数据*)
			IF ABS(Axis_QJ.QJ_AxisState.rActPosition-Axis_QJ.QJ_AxisCmd.AxisPara.rAbsPosition)<1 AND Axis_QJ.QJ_AxisState.bStandStill THEN
				WorkStation_TCP.PLC_SEND1.m_nMoveState:=1; 			//send [9]
				Step_StandardCT:=70;				//自动扫描
			ELSE
				WorkStation_TCP.PLC_SEND1.m_nMoveState:=0; 			//send [9]	//0-准备过程中 1-准备完成 2-曝光中 3-本次扫描结束
			END_IF
			
		(*-------------------------手动扫描-----------------------------*)	
		200://中间状态清零
			WorkStation_TCP.PLC_SEND1.m_nMoveState:=0; //send [9]	//0-准备过程中 1-准备完成 2-曝光中 3-本次扫描结束
			Axis_XZ.XZ_AxisCmd.bAbs:=FALSE;
			Step_StandardCT:=210;
			
		210://7灯闪烁，机架运动到目标位置
			(*1.发送给上位机的数据*)
			WorkStation_TCP.PLC_SEND1.m_nMoveState:=0; //send [9]	//0-准备过程中 1-准备完成 2-曝光中 3-本次扫描结束
			
			(*2.7灯闪烁*)
			LampCmd7:=E_LampCmd.慢闪;
			WorkStation_TCP.PLC_SEND1.m_nFocus:=7;	//按键提示0228
			
			(*3.旋转轴运动到目标位置*)
			Axis_XZ.XZ_AxisCmd.AxisPara.rAbsPosition:=LIMIT(-4,WorkStation_TCP.PLC_RECV1.m_nRotateBegin,363);
			Axis_XZ.XZ_AxisCmd.AxisPara.rAbsVelocity:=XZ_Velocity;
			
			IF WorkStation_TCP.PLC_RECV1.m_nSocketType=1 THEN
				Axis_XZ.XZ_AxisCmd.bAbs:=TRUE;
			END_IF;
			
			(*4.到位后2秒跳转*)
			IF ABS(Axis_XZ.XZ_AxisState.rActPosition-WorkStation_TCP.PLC_RECV1.m_nRotateBegin)<1 AND Axis_XZ.XZ_AxisState.bStandStill THEN
				Step_StandardCT:=220;	
			END_IF
		
		220://中间状态清零
			Axis_XZ.XZ_AxisCmd.bAbs:=FALSE;
			Axis_QJ.QJ_AxisCmd.bAbs:=FALSE;
			Step_StandardCT:=230;
			
		230://用户按7键，床自动走到预设位置
			(*1.按7键关闭7灯*)
			IF CTBOX_RS232.CTBOX_KEY_Manual THEN
				LampCmd7:=E_LampCmd.关闭;
				WorkStation_TCP.PLC_SEND1.m_nFocus:=0;	//关闭按键提示0228
			END_IF
			
			(*2.触发床运动*)
			R_TRIG_G2(CLK:=CTBOX_RS232.CTBOX_KEY_Manual , Q=> );
			Axis_QJ.QJ_AxisCmd.AxisPara.rAbsPosition:=LIMIT(0,WorkStation_TCP.PLC_RECV1.m_fScanTop,900);
			Axis_QJ.QJ_AxisCmd.bAbs:=R_TRIG_G2.Q;
			
			(*3.跳转指令*)
			IF ABS(Axis_QJ.QJ_AxisState.rActPosition-WorkStation_TCP.PLC_RECV1.m_fScanTop)<1 AND (LampCmd7=E_LampCmd.关闭) THEN //保证必须按下7键
				WorkStation_TCP.PLC_SEND1.m_nMoveState:=1; //send [9]	//0-准备过程中 1-准备完成 2-曝光中 3-本次扫描结束
			ELSE
				WorkStation_TCP.PLC_SEND1.m_nMoveState:=0; //send [9]	//0-准备过程中 1-准备完成 2-曝光中 3-本次扫描结束
			END_IF
			
			(*4.延迟跳转，保证send [9]发送*)
			TON_CT_G[11](IN:=(WorkStation_TCP.PLC_SEND1.m_nMoveState=1) , PT:=T#1100MS , Q=> , ET=> );
			IF TON_CT_G[11].Q THEN
				Step_StandardCT:=60;
			END_IF
	END_CASE
END_ACTION

ACTION _a_ShutDown_entry_1:

	(**)
	GVL_State.iPLC_State:=340;
	(*伺服电机停止*)
	Axis_XZ.XZ_AxisCmd.bStop:=TRUE;
	Axis_QJ.QJ_AxisCmd.bStop:=TRUE;
	
	(*射线停止输出*)
	Entity_IO.bXaryTwo:=FALSE;
	Entity_IO.bXaryOne:=FALSE;
	Entity_IO.bXaryFlu:=FALSE;
	Step_ShutDown:=0;
	bOver:=FALSE;
END_ACTION

TRANSITION T_JUMP_IDLE:


	(*跳转到待机指令*)
	(*1.手动终止扫描，上位机发送终止扫描，扫描结束*)
	TON_StopScan.Q 
	OR (WorkStation_TCP.PLC_RECV1.m_nControlState>=1 AND WorkStation_TCP.PLC_RECV1.m_nSocketType=1)
	OR GVL_SCAN.bJumpScan;
END_TRANSITION

ACTION _a_StaticDR_exit:

	Entity_IO.bTriggerOut:=FALSE;
	Entity_IO.bXaryOne:=FALSE;
	Entity_IO.bXaryTwo:=FALSE;
	Step_StaticDR:=00;
	TOF_DR111(IN:=FALSE);
	WorkStation_TCP.PLC_SEND1.m_nFocus:=0;					//按键关闭
END_ACTION

ACTION _a_Emergercy_active_1:


(*急停工作模式*)

(*1.所有电机下使能,升降电机禁止运动*)
	Axis_XZ.XZ_AxisCmd.bPower:=FALSE;//上使能
	Axis_QJ.QJ_AxisCmd.bPower:=FALSE;//上使能

	Motor_SJ(Enable:= FALSE);

(*2.射线源停止出束，一二档信号失能*)
	Entity_IO.bXaryTwo:=FALSE;
	Entity_IO.bXaryOne:=FALSE;
	Entity_IO.bXaryFlu:=FALSE;
END_ACTION

ACTION _a_StaticCT_active:


	CASE Step_Scout OF
		0:	//初始化准备流程
			(*1.给上位机发送的数据*)
			WorkStation_TCP.PLC_SEND1.m_nMoveState:=0;			//send[9]
			
			(*2.运动准备数据*)
			(*2.1 写入旋转速度参数*)
			Axis_XZ.XZ_AxisCmd.AxisPara.rAbsVelocity:=36;//定位像扫描按照设定速度运动
			Axis_XZ.XZ_AxisCmd.bAbs	:=FALSE;
			bScoutLast 				:=FALSE;
			
			(*3.//运动过程中变量复位标志*)
			FOR i:=1 TO 50 BY 1 DO 
				TON_CT_J[i](IN:= FALSE);
			END_FOR
		
			(*4.跳转*)
			Step_Scout:=10;

		10://开启运动
			(*1.给上位机发送的数据*)
			WorkStation_TCP.PLC_SEND1.m_nExpStates	:=1;//为曝光状态，枚举值，0:idle（空闲） 1:prep（训机） 2: ready（训机结束，准备完成，可以出束） 3: XrayOn（出射线） 4:XrayOff（关射线） 5 error；
			WorkStation_TCP.PLC_SEND1.m_nMoveState	:=0;//起始、终止状态， 默认值-1， 0为当前扫描方案（与常规意义不同，注意区别）处于准备好状态，可以准备扫描；1为当前扫描方案结束，运动过程中值为-1
			WorkStation_TCP.PLC_SEND1.m_nScanProType:=2;//执行扫描方案的类型，0为自动扫描，1为手动扫描，2为无设置意义的值，默认值为2
	
			(*2.旋转轴运动*)
			TON_CT_J[1](IN:= TRUE, PT:=T#500MS);
			Axis_XZ.XZ_AxisCmd.bAbs:=TON_CT_J[1].Q;
			Axis_XZ.XZ_AxisCmd.AxisPara.rAbsPosition:=LIMIT(-4,WorkStation_TCP.PLC_RECV1.m_nRotateBegin,363);

			(*3.跳转下一个步骤*)	
			IF  ABS(Axis_XZ.XZ_AxisState.rActPosition-WorkStation_TCP.PLC_RECV1.m_nRotateBegin)<=1 AND Axis_XZ.XZ_AxisState.bStandStill THEN(*OR Axis_XZ.XZ_AxisState.bStandStill*)
				Step_Scout:=20;
			END_IF
				
		20://射线源参数写入成功标志
			(*1.状态复位*)
			TON_CT_J[1](IN:=FALSE);
			Axis_XZ.XZ_AxisCmd.bAbs:=FALSE;
			
			(*2.等待射线源参数成功写入*)
			IF DT_Xray.ExpPara_Step=66 THEN		
				Step_Scout:=30;
			END_IF

		30: //开启7灯闪烁
			(*1.给上位机数据*)
			WorkStation_TCP.PLC_SEND1.m_nMoveState:=1;	 //send[9]
			
			(*2.7灯闪烁*)
			LampCmd7:=E_LampCmd.慢闪;
			WorkStation_TCP.PLC_SEND1.m_nFocus:=7;		//按键提示0228
			
			(*3.跳转*)
			TON_CT_J[2](IN:=TRUE , PT:=T#1S);
			IF TON_CT_J[2].Q THEN
				Step_Scout:=40;
			END_IF
		
		40://等待用户按7键。此时7灯一直在闪烁
			(*1.发送上位机状态*)
			IF CTBOX_RS232.CTBOX_KEY_Manual THEN
				WorkStation_TCP.PLC_SEND1.m_nScanProType:=1;//执行扫描方案的类型，0为自动扫描，1为手动扫描，2为无设置意义的值，默认值为2
			END_IF
			
			(*2.7灯关闭*)
			TON_CT_J[3](IN:=(WorkStation_TCP.PLC_SEND1.m_nScanProType=1) , PT:=T#100MS , Q=> , ET=> );
			IF TON_CT_J[3].Q THEN
				LampCmd7:=E_LampCmd.关闭;  					//7灯关闭
				WorkStation_TCP.PLC_SEND1.m_nFocus:=0;		//关闭按键提示0228
			END_IF

			(*3.跳转*)
			TON_CT_J[4](IN:= (WorkStation_TCP.PLC_SEND1.m_nScanProType=1), PT:=T#1S , Q=> , ET=> );
			IF TON_CT_J[4].Q THEN
				Step_Scout:=50;
			END_IF
			
		50://中间状态清零，特别是从80跳转过来的变量清零
			FOR i:=1 TO 50 BY 1 DO 
				TON_CT_J[i](IN:= FALSE);
			END_FOR
			R_CT_J1(CLK:= FALSE);
			Entity_IO.bXaryOne:=FALSE;Entity_IO.bXaryTwo:=FALSE;
			Axis_QJ.QJ_AxisCmd.bAbs:=FALSE;
			Axis_XZ.XZ_AxisCmd.bAbs:=FALSE;
			
			(*2.射线源参数写完完毕*)
			IF  DT_Xray.ExpPara_Step=66  THEN
				Step_Scout:=55;
			END_IF;	
			
		55://增加上位机扫描方案延迟
			DelayTime:=T#1MS*WorkStation_TCP.PLC_RECV1.m_nDelayTime;
			TON_CT_J[13](IN:=TRUE , PT:=DelayTime , Q=> , ET=> );
			IF TON_CT_J[13].Q THEN
				Step_Scout:=60;
			END_IF

		60:
			(*1.开启曝光指令*)
			Entity_IO.bXaryOne:=TRUE;		//开启一档
			Entity_IO.bXaryTwo:=TRUE;		//开启二档
			
			(*2.判断是否最后一次扫描标志位*)
			IF WorkStation_TCP.PLC_RECV1.m_nLastMsg=1 THEN bScoutLast := TRUE;
			ELSE bScoutLast := FALSE;
			END_IF
			
			(*3.获取此次曝光时间*)
			TimeScoutExp:=REAL_TO_TIME(WorkStation_TCP.PLC_RECV1.m_nMS)+T#1MS;

			(*3.跳转指令*)
			IF DT_Xray.RadExp_Step>=10 THEN  //此时射线源收到  =25
				Step_Scout:=68;
			END_IF 
			
			(*4.一二档信号超时报警，射线源30秒连续开启曝光会报警*)
			TON_CT_J[5](IN:=Entity_IO.bXaryTwo , PT:=T#30S , Q=> , ET=> );
			IF TON_CT_J[5].Q THEN
				Step_Scout:=44;	
			END_IF
			
			(*5.触发一张采图*)
			R_CT_J1(CLK:= Entity_IO.bXaryTwo, Q=>Entity_IO.bTriggerOut );
			
		68:
			Step_Scout:=70;
			R_CT_J1(CLK:= FALSE);	
			Entity_IO.bTriggerOut:=FALSE;
			
		44:
			Entity_IO.bXaryOne	:=FALSE;
			Entity_IO.bXaryTwo	:=FALSE;
			GVL_SCAN.bJumpScan	:=TRUE;		//结束扫描，射线源超时报警了，EL019，结束扫描
			Step_Scout			:=44;	

		70://固定位置直接采图，曝光指令在DT_Xray任务里
			TON_CT_J[5](IN:=FALSE);	//复位
	
			(*1.发送给上位机的数据*)
			WorkStation_TCP.PLC_SEND1.m_nMoveState	:=2;			//send[9]//0-准备过程中 1-准备完成 2-曝光中 3-本次扫描结束	
			WorkStation_TCP.PLC_SEND1.m_nScanProType:=2;			//send[16]
			
			(*2.开启触发信号采集出图，仅触发一次*)
			TON_CT_J[6](IN:=TRUE,PT:=TimeScoutExp);

			F_TRIG_S(CLK:=Entity_IO.bXaryTwo , Q=> );
			(*3.曝光结束，跳出*)
			IF DT_Xray.RadExp_Step=66 AND TON_CT_J[6].Q THEN
				Step_Scout:=78;	
			END_IF
			
		78:
			Entity_IO.bTriggerOut:=FALSE;
			TON_CT_J[11](IN:=TRUE,PT:=T#100MS);
			IF TON_CT_J[11].Q THEN
				Step_Scout:=80;	
			END_IF
		
		80://判断是否最后一次扫描，如是，直接跳到待机模式，如果不是，接着定位扫描 ，第一次定位像和第二次定位像不一样，增加了床的运动
			(*1.运动变量复位*)
			Entity_IO.bXaryOne:=FALSE;
			Entity_IO.bXaryTwo:=FALSE;
			Axis_QJ.QJ_AxisCmd.bAbs:=FALSE;
			Axis_XZ.XZ_AxisCmd.bAbs:=FALSE;	
			Entity_IO.bTriggerOut:=FALSE;
			F_TRIG_S(CLK:=Entity_IO.bXaryTwo , Q=>Entity_IO.bTriggerOut );

			(*2.给上位机发送数据，不能太快*)
			TON_CT_J[7](IN:=TRUE , PT:=T#1600MS , Q=> , ET=> );	//留些时间给上位机发送本次扫描结束方案标志
			
			IF DT_Xray.RadExp_Step=77 THEN 
				WorkStation_TCP.PLC_SEND1.m_nMoveState:=3;			//send[9] //0-准备过程中 1-准备完成 2-曝光中 3-本次扫描结束
			END_IF;
			
			(*3.判断师傅最后一次扫描*)
			IF TON_CT_J[7].Q THEN
				IF (WorkStation_TCP.PLC_RECV1.m_nCircleIndex+1)>=(WorkStation_TCP.PLC_RECV1.m_nCircleCount) AND bScoutLast AND DT_Xray.RadExp_Step=77 THEN 	//用于区分自动扫是否最后一次，此时=1，=1都等于1
					GVL_SCAN.bJumpScan:=TRUE;
				END_IF;
			END_IF
			
			(*4.不是最后一次，收到下一次命令，继续扫*)
			IF WorkStation_TCP.PLC_RECV1.m_nSocketType=1 AND DT_Xray.RadExp_Step=77 THEN 	//增加第二次运动判断，m_nSocketType=1 
				Step_Scout:=90;
			END_IF
			
		90://上位机选择移动床位置，机架根据命令运动到位
			(*1.前进电机运动*)
			Axis_QJ.QJ_AxisCmd.AxisPara.rAbsPosition:=LIMIT(0,WorkStation_TCP.PLC_RECV1.m_fScanTop,900);
			Axis_QJ.QJ_AxisCmd.AxisPara.rAbsVelocity:=50; //单位mm/s
			TON_CT_J[8](IN:=TRUE , PT:=T#500MS );
			Axis_QJ.QJ_AxisCmd.bAbs:=TON_CT_J[8].Q;
			
			(*2.旋转电机运动*)
			Axis_XZ.XZ_AxisCmd.AxisPara.rAbsPosition:=LIMIT(-4,WorkStation_TCP.PLC_RECV1.m_nRotateBegin,363);
			TON_CT_J[9](IN:=TRUE , PT:=T#500MS );
			Axis_XZ.XZ_AxisCmd.bAbs:=TON_CT_J[9].Q;
			
			(*3.给上位机发送的数据*)
			IF ABS(Axis_QJ.QJ_AxisState.rActPosition-WorkStation_TCP.PLC_RECV1.m_fScanTop)<1 AND ABS(Axis_XZ.XZ_AxisState.rActPosition-WorkStation_TCP.PLC_RECV1.m_nRotateBegin)<1 THEN
				WorkStation_TCP.PLC_SEND1.m_nMoveState:=1;		//send[9] //0-准备过程中 1-准备完成 2-曝光中 3-本次扫描结束	
			ELSE
				WorkStation_TCP.PLC_SEND1.m_nMoveState:=0;		//send[9] //0-准备过程中 1-准备完成 2-曝光中 3-本次扫描结束	
			END_IF
			
			(*4.跳转指令*)
			TON_CT_J[10](IN:=ABS(Axis_QJ.QJ_AxisState.rActPosition-WorkStation_TCP.PLC_RECV1.m_fScanTop)<1 
					AND ABS(Axis_XZ.XZ_AxisState.rActPosition-WorkStation_TCP.PLC_RECV1.m_nRotateBegin)<1
					AND Axis_XZ.XZ_AxisState.bStandStill AND Axis_QJ.QJ_AxisState.bStandStill, 
					PT:=T#2S , Q=> , ET=> );//给你2秒走到位
			IF TON_CT_J[10].Q THEN
				Step_Scout:=50;
			END_IF
		
	END_CASE
END_ACTION

ACTION _a_Idle_exit:


	Step_Idle:=0;
	
	LampCmd5:=E_LampCmd.关闭;
	LampCmd6:=E_LampCmd.关闭;
	LampCmd7:=E_LampCmd.关闭;
	LampCmd8:=E_LampCmd.关闭;
END_ACTION

TRANSITION T_StaticDR:

(*进入dr扫描*)
	WorkStation_TCP.PLC_RECV1.m_nSocketType=1 AND WorkStation_TCP.PLC_RECV1.m_nExpId=1
END_TRANSITION

TRANSITION T_DynamicsDR:

(*进入动态DR扫描*)
	WorkStation_TCP.PLC_RECV1.m_nSocketType=1 AND WorkStation_TCP.PLC_RECV1.m_nExpId=2
END_TRANSITION

ACTION _a_Idle_entry:


	Step_Idle:=0; //
	bPulseOneStop:=TRUE;
	
	GVL_SCAN.bJumpScan:=FALSE;
	
	Axis_XZ.XZ_AxisCmd.bAbs:=FALSE;
	Axis_QJ.QJ_AxisCmd.bAbs:=FALSE;
	
	Axis_QJ.QJ_AxisCmd.bStop:=FALSE;
	Axis_XZ.XZ_AxisCmd.bStop:=FALSE;
		
	Axis_XZ.XZ_AxisCmd.bReset:=FALSE;
	Axis_QJ.QJ_AxisCmd.bReset:=FALSE;
	
	
	WorkStation_TCP.PLC_SEND1.m_nFocus:=0;//按键提示

	Step_CBCT:=0;
	Step_Scout:=0;
END_ACTION

ACTION _a_StaticCT_entry:


Step_Scout:=0; 

GVL_State.iPLC_State:=220;
END_ACTION

TRANSITION T_CT:

WorkStation_TCP.PLC_RECV1.m_nSocketType=1 AND (WorkStation_TCP.PLC_RECV1.m_nExpId>=3 AND  WorkStation_TCP.PLC_RECV1.m_nExpId<=6)
END_TRANSITION

ACTION _a_SelfCheck_exit:


//Axis_QJ.QJ_AxisCmd.bSetHomePara:=TRUE;

//Axis_XZ.XZ_AxisCmd.bSetHomePara:=TRUE;
END_ACTION

ACTION _a_Error_entry:

	bErrorReset:=TRUE;
	TON_Error(IN:=FALSE);
END_ACTION

TRANSITION T_QuickCT:


(*进入快速扫描*)
	WorkStation_TCP.PLC_RECV1.m_nSocketType=1 AND WorkStation_TCP.PLC_RECV1.m_nExpId=6
END_TRANSITION

ACTION _a_Error_active:
(*电机进行复位操作*)	
	IF bErrorReset THEN	
		IF (Axis_XZ.XZ_AxisState.bAxisErr OR Axis_XZ.XZ_AxisState.bErrStop) AND  TON_Error1.Q THEN
			Axis_XZ.XZ_AxisCmd.bReset:=TRUE;
		ELSE
			;		
		END_IF
		
		IF (Axis_QJ.QJ_AxisState.bAxisErr  OR  Axis_QJ.QJ_AxisState.bErrStop) AND  TON_Error1.Q THEN
			Axis_QJ.QJ_AxisCmd.bReset:=TRUE;
		ELSE
			;		
		END_IF
		
		IF Axis_XZ.XZ_AxisState.bAxisErr=FALSE AND  Axis_XZ.XZ_AxisState.bErrStop=FALSE AND Axis_QJ.QJ_AxisState.bAxisErr=FALSE  AND  Axis_QJ.QJ_AxisState.bErrStop=FALSE THEN
			bErrorReset:=FALSE;
		END_IF
	ELSE
		Axis_QJ.QJ_AxisCmd.bReset:=FALSE;
		Axis_XZ.XZ_AxisCmd.bReset:=FALSE;
	END_IF
	
	(*延迟2秒输出*)
	TON_Error(IN:=TRUE , PT:=T#1S , Q=> , ET=> );
	IF TON_Error.Q THEN
		GVL_State.iPLC_State:=310;
	END_IF
	
	TON_Error1(IN:= bErrorReset, PT:= T#2S, Q=> , ET=> );
END_ACTION

ACTION _a_HighDefinCT_active:

	CASE Step_CBCT OF 
		0:	//初始化准备流程
			(*1.给上位机发送的数据*)
			WorkStation_TCP.PLC_SEND1.m_nMoveState:=0;			//send[9] //0-准备过程中 1-准备完成 2-曝光中 3-本次扫描结束 
			bCBCTLast		:=FALSE;
			
			(*2.运动准备数据*)
			(*2.1 写入旋转速度参数*)
			IF WorkStation_TCP.PLC_RECV1.m_fSecondPerCicle<>0 THEN//避免除零
				Axis_XZ.XZ_AxisCmd.AxisPara.rAbsVelocity:=(LIMIT(360/300 ,360/WorkStation_TCP.PLC_RECV1.m_fSecondPerCicle ,360/20));
				XZ_Velocity:=LIMIT(360/300 ,360/(WorkStation_TCP.PLC_RECV1.m_fSecondPerCicle) ,360/20);
			ELSE
				Axis_XZ.XZ_AxisCmd.AxisPara.rAbsVelocity:=8;
			END_IF;
			
			(*3.中间变量复位*)
			FOR i:=1 TO 50 BY 1 DO 
				TON_CT_G[i](IN:= FALSE);
			END_FOR
			Axis_XZ.XZ_AxisCmd.bAbs		:=FALSE;
			Axis_QJ.QJ_AxisCmd.bAbs		:=FALSE;
			Step_CBCT:=10;
				
		10://按5键，移动床到预设位置，松开即停，机架直接到预设位置
			(*1.发送给上位机的数据*)
			WorkStation_TCP.PLC_SEND1.m_nExpStates	:=1;		//0-准备过程中 1-准备完成 2-曝光中 3-本次扫描结束	
			WorkStation_TCP.PLC_SEND1.m_nMoveState	:=0;		//起始、终止状态， 默认值0， 1为当前扫描方案处于准备好状态，可以准备扫描；2为当前扫描方案结束，运动过程中值为0
			WorkStation_TCP.PLC_SEND1.m_nScanProType:=2;		//扫描方案类型 , 1-手动，0-自动. 
			
			(*2.旋转轴直接运动到目标位置*)
			Axis_XZ.XZ_AxisCmd.AxisPara.rAbsPosition	:=LIMIT(-3,WorkStation_TCP.PLC_RECV1.m_nRotateBegin,363);
			Axis_XZ.XZ_AxisCmd.AxisPara.rAbsVelocity	:=18;
			TON_CT_G[1](IN:=TRUE , PT:=T#500MS);
			Axis_XZ.XZ_AxisCmd.bAbs						:=TON_CT_G[1].Q;
			
			(*3.前进轴运动*)
			R_TRIG_G1(CLK:= CTBOX_RS232.CTBOX_KEY_MoveDistance, Q=> );//触发运动
			F_TRIG_G1(CLK:= CTBOX_RS232.CTBOX_KEY_MoveDistance, Q=> );//触发停止
			
			Axis_QJ.QJ_AxisCmd.bAbs	:=R_TRIG_G1.Q;
			Axis_QJ.QJ_AxisCmd.AxisPara.rAbsPosition	:=LIMIT(0,WorkStation_TCP.PLC_RECV1.m_fScanTop,900);
			Axis_QJ.QJ_AxisCmd.bStop:=F_TRIG_G1.Q;
			
			(*4.5灯逻辑处理*)
			IF ABS(Axis_QJ.QJ_AxisState.rActPosition-WorkStation_TCP.PLC_RECV1.m_fScanTop)>=1 THEN
				LampCmd5:=E_LampCmd.慢闪;
				WorkStation_TCP.PLC_SEND1.m_nFocus:=5;			//按键提示0228
			ELSE
				LampCmd5:=E_LampCmd.关闭;
				WorkStation_TCP.PLC_SEND1.m_nFocus:=0;			//关闭按键提示0228
			END_IF
			
			(*5.跳转*)
			TON_CT_G[2](IN:=ABS(Axis_QJ.QJ_AxisState.rActPosition-WorkStation_TCP.PLC_RECV1.m_fScanTop)<1 
				AND ABS(Axis_XZ.XZ_AxisState.rActPosition-WorkStation_TCP.PLC_RECV1.m_nRotateBegin)<1 
				AND Axis_XZ.XZ_AxisState.bStandStill AND Axis_QJ.QJ_AxisState.bStandStill, PT:=T#100MS);
			IF TON_CT_G[2].Q THEN  
				Step_CBCT:=20;
			END_IF
			
		20:	//射线源参数写入成功标志
			(*1.变量复位*)
			LampCmd5:=E_LampCmd.关闭;
			Axis_XZ.XZ_AxisCmd.bAbs		:=FALSE;
			Axis_QJ.QJ_AxisCmd.bAbs		:=FALSE;
			Axis_QJ.QJ_AxisCmd.bStop	:=FALSE;
			
			(*2.射线源参数写入正常完毕*)
			IF DT_Xray.FluPara_Setp=66 THEN
				Step_CBCT:=30;
			END_IF
			
		30:	//7灯和8灯开始慢闪
			(*1.给上位机发送的数*)
			WorkStation_TCP.PLC_SEND1.m_nMoveState	:=1;		//起始、终止状态， 默认值0， 1为当前扫描方案处于准备好状态
			WorkStation_TCP.PLC_SEND1.m_nFocus		:=8;		//按键提示0228
			
			(*2.CTBOX灯的状态*)
			LampCmd7:=E_LampCmd.慢闪;
			LampCmd8:=E_LampCmd.慢闪;
			
			TON_CT_G[3](IN:=TRUE , PT:=T#600MS);
			IF TON_CT_G[3].Q THEN
				Step_CBCT:=40;
			END_IF
		
		40://用户选择自动扫描或手动扫描
			IF CTBOX_RS232.CTBOX_KEY_Auto=FALSE AND CTBOX_RS232.CTBOX_KEY_Manual THEN
				WorkStation_TCP.PLC_SEND1.m_nScanProType:=1;								//扫描方案类型 , 1-手动，0-自动. 
				bCBCT_AUTO_Manual:=TRUE;
			ELSIF CTBOX_RS232.CTBOX_KEY_Auto AND CTBOX_RS232.CTBOX_KEY_Manual=FALSE THEN
				WorkStation_TCP.PLC_SEND1.m_nScanProType:=0;								//扫描方案类型 , 1-手动，0-自动. 
				bCBCT_AUTO_Manual:=FALSE;
			ELSIF CTBOX_RS232.CTBOX_KEY_Auto=FALSE AND CTBOX_RS232.CTBOX_KEY_Manual=FALSE THEN
				;
			ELSIF CTBOX_RS232.CTBOX_KEY_Auto AND CTBOX_RS232.CTBOX_KEY_Manual THEN
				;
			END_IF
			
			IF (CTBOX_RS232.CTBOX_KEY_Auto AND CTBOX_RS232.CTBOX_KEY_Manual=FALSE) OR CTBOX_RS232.CTBOX_KEY_Manual AND CTBOX_RS232.CTBOX_KEY_Auto=FALSE THEN
				Step_CBCT:=50;
			END_IF
			
		50://7和8灯关闭 
			(*1.给上位机发送的数据*)
			WorkStation_TCP.PLC_SEND1.m_nFocus:=0;	//关闭按键提示0228
			
			(*2.CTBOX灯关闭*)
			LampCmd7:=E_LampCmd.关闭;
			LampCmd8:=E_LampCmd.关闭;
			
			(*3.获取当前编码器数值*)
			iStartTrigger1:=Entity_IO.iEncoderPulse;//只赋值一次
			
			(*4.跳转*)
			TON_CT_G[4](IN:= TRUE, PT:=T#1S);
			IF TON_CT_G[4].Q THEN
				Step_CBCT:=60;
			END_IF
			
		60://扫描中间态，给跳转用的
			(*1.变量复位*)
			FOR i:=1 TO 50 BY 1 DO 
				TON_CT_G[i](IN:= FALSE);
			END_FOR
			Axis_QJ.QJ_AxisCmd.bAbs:=FALSE;//复位前进轴
			Axis_XZ.XZ_AxisCmd.bAbs:=FALSE;//复位旋转轴
			iActNumPulse:=0;
			Step_CBCT:=65;
			
		65://增加上位机扫描方案延迟
			DelayTime:=T#1MS*WorkStation_TCP.PLC_RECV1.m_nDelayTime;
			TON_CT_G[17](IN:=TRUE , PT:=DelayTime , Q=> , ET=> );
			IF TON_CT_G[17].Q THEN
				Step_CBCT:=70;
			END_IF
			
		70:
			(*1.发送给上位机的数据*)
			WorkStation_TCP.PLC_SEND1.m_nMoveState	:=1;	//send[9]
			WorkStation_TCP.PLC_SEND1.m_nScanProType:=2;	//send[16]
			
			(*2.射线源参数写入成功，开启透视*)
			IF DT_Xray.FluPara_Setp=66 THEN  //保证写入参数
				Entity_IO.bXaryFlu:=TRUE;//开启透视
			END_IF;
			
			(*3.判断是否最后一次扫描*)
			IF WorkStation_TCP.PLC_RECV1.m_nLastMsg=1 THEN
				bCBCTLast := TRUE;
			ELSE
				bCBCTLast := FALSE;
			END_IF
			
			(*4.获取上位机发送的采样率*)//
			iSamplingRate:=UDINT_TO_UINT(WorkStation_TCP.PLC_RECV1.m_nSamplingRate);//采样率，有4个选项：2400帧/圈；1200帧/圈；600帧/圈,360帧/圈
			
			(*5.处理多少个脉冲输出一个trigger*)
			CASE iSamplingRate OF 
				360:iHopePulse:=360;
				600:iHopePulse:=216;
				1200:iHopePulse:=108;
				2400:iHopePulse:=54;
				ELSE iHopePulse:=360;
			END_CASE

			(*6.跳转指令*)
			TON_CT_G[5](IN:=TRUE,PT:=T#600MS);
			IF TON_CT_G[5].Q AND Entity_IO.bXaryFlu THEN
				Step_CBCT:=80;
			END_IF
			
			(*7.计数清零,多协议扫描清零用*)
			iActNumPulse:=0;
		74:
			Entity_IO.bXaryFlu:=FALSE;
			GVL_SCAN.bJumpScan:=TRUE;		//结束扫描，射线源超时报警了，EL019，结束扫描
			Step_CBCT:=74;
			
		80://第一次自动扫描
			(*1.给上位机发送的数*)
			WorkStation_TCP.PLC_SEND1.m_nMoveState	:=2;
			WorkStation_TCP.PLC_SEND1.m_nScanProType:=2;

			(*2.触发旋转轴运动*)
			Axis_XZ.XZ_AxisCmd.AxisPara.rAbsPosition:=LIMIT(-3,WorkStation_TCP.PLC_RECV1.m_nRotateEnd,363);
			Axis_XZ.XZ_AxisCmd.AxisPara.rAbsVelocity:=XZ_Velocity;
			TON_CT_G[6](IN:=TRUE , PT:=T#500MS );
			Axis_XZ.XZ_AxisCmd.bAbs:=TON_CT_G[6].Q;
					
			(*4.开启允许采图指令*)
			(*4.1.获取旋转编码器的数值*)
			EncoderNum1:=Entity_IO.iEncoderPulse;
			(*4.2处理相对脉冲来作为触发*)
			DB_EncoderNum1:=ABS(EncoderNum1-iStartTrigger1);
			iValidTrigger:=DINT_TO_UINT(DB_EncoderNum1 MOD iHopePulse);
			
			IF (iActNumPulse)<=(iSamplingRate+2) THEN
				IF (iValidTrigger)<=1*iHopePulse / 2 THEN  	//1/3的占空比，这个时间要和上位机下发的扫描时间对应 24秒一圈，30帧频 目前探测器达不到30帧7、8
					Entity_IO.bTriggerOut:=TRUE;
				ELSE
					Entity_IO.bTriggerOut:=FALSE;
				END_IF
			ELSE
				Entity_IO.bTriggerOut:=FALSE;
			END_IF;
			
			(*4.3 计数器计算*)
			F_TRIG_G2(CLK:=Entity_IO.bTriggerOut , Q=>);
			IF F_TRIG_G2.Q THEN iActNumPulse:=iActNumPulse+1;END_IF;

			(*5.跳转,到达终止角度*)
			TON_CT_G[7](IN:= ABS(Axis_XZ.XZ_AxisState.rActPosition-WorkStation_TCP.PLC_RECV1.m_nRotateEnd)<1 AND Axis_XZ.XZ_AxisState.bStandStill, PT:=T#100MS , Q=> , ET=> );	
			IF TON_CT_G[7].Q THEN
				Step_CBCT:=89;
			END_IF
			
			(*6.透视信号超时报警，射线源30秒连续开启曝光会报警*)
			TON_CT_G[8](IN:=Entity_IO.bXaryFlu , PT:=T#3M , Q=> , ET=> );
			IF TON_CT_G[8].Q THEN
				Step_CBCT:=74;	
			END_IF
		89:
			Entity_IO.bTriggerOut	:=FALSE;
			TON_CT_G[15](IN:=TRUE , PT:=T#500MS , Q=> , ET=> );
			IF 	TON_CT_G[15].Q THEN
				Step_CBCT:=90;
			END_IF
			
			
		90://出射线状态结束，采集射线源状态机信息
			(*1.关闭透视信号*)
			Entity_IO.bXaryFlu		:=FALSE;
			Axis_XZ.XZ_AxisCmd.bAbs	:=FALSE;
			(*2.跳转*)
			
			IF GVL_State.iXray_State=40 THEN	//DT射线源增加状态 ,回到待机状态 
				Step_CBCT:=100;
			END_IF
			
		100://中间变量清零1070
			(*1.给上位机发送的数据*)
			WorkStation_TCP.PLC_SEND1.m_nMoveState:=3; //send [9]
			
			(*2.判断是否最后一次扫描*)
			TON_CT_G[9](IN:=TRUE , PT:=T#1S , Q=> , ET=> );
			IF TON_CT_G[9].Q THEN
				IF (WorkStation_TCP.PLC_RECV1.m_nCircleIndex+1)>=(WorkStation_TCP.PLC_RECV1.m_nCircleCount) AND bCBCTLast THEN //最后一次扫描退出
					GVL_SCAN.bJumpScan:=TRUE;
				END_IF
			END_IF
		
			(*3.不是最后一次增加跳转判断增加跳转接着扫*)
			IF WorkStation_TCP.PLC_RECV1.m_nSocketType=1 THEN 	//增加第二次运动判断，m_nSocketType=1 
				Step_CBCT:=110;
			END_IF
			
		110:
			FOR i:=1 TO 30 BY 1 DO 
				TON_CT_G[i](IN:= FALSE);
			END_FOR
			//CBCT下的自动扫还是手动扫，根据上位机命令
			IF WorkStation_TCP.PLC_RECV1.m_nScanMoveType=1 THEN
				Step_CBCT:=200;		//手动扫描
			ELSE
				Step_CBCT:=120;		//自动扫描
			END_IF
		 
		120://开启自动扫描
			(*1.前进轴自动运动*)
			TON_CT_G[10](IN:=TRUE , PT:=T#300MS , Q=> , ET=> );
			Axis_QJ.QJ_AxisCmd.AxisPara.rAbsPosition:=LIMIT(0,WorkStation_TCP.PLC_RECV1.m_fScanTop,900);
			Axis_QJ.QJ_AxisCmd.bAbs:=TON_CT_G[10].Q;
			
			(*2.给上位机发送的数据*)
			IF ABS(Axis_QJ.QJ_AxisState.rActPosition-WorkStation_TCP.PLC_RECV1.m_fScanTop)<1 AND Axis_QJ.QJ_AxisState.bStandStill THEN
				WorkStation_TCP.PLC_SEND1.m_nMoveState:=1; 			//send [9]
				Step_CBCT:=70;				//自动扫描
			ELSE
				WorkStation_TCP.PLC_SEND1.m_nMoveState:=0; 			//send [9]	//0-准备过程中 1-准备完成 2-曝光中 3-本次扫描结束
			END_IF
			
		(*-------------------------手动扫描-----------------------------*)	
		200://中间状态清零
			WorkStation_TCP.PLC_SEND1.m_nMoveState:=0; //send [9]	//0-准备过程中 1-准备完成 2-曝光中 3-本次扫描结束
			Axis_XZ.XZ_AxisCmd.bAbs:=FALSE;
			Step_CBCT:=210;
			
		210://7灯闪烁，机架运动到目标位置
			(*1.发送给上位机的数据*)
			WorkStation_TCP.PLC_SEND1.m_nMoveState:=0; //send [9]	//0-准备过程中 1-准备完成 2-曝光中 3-本次扫描结束
			
			(*2.7灯闪烁*)
			LampCmd7:=E_LampCmd.慢闪;
			WorkStation_TCP.PLC_SEND1.m_nFocus:=7;	//按键提示0228
			
			(*3.旋转轴运动到目标位置*)
			Axis_XZ.XZ_AxisCmd.AxisPara.rAbsPosition:=LIMIT(-4,WorkStation_TCP.PLC_RECV1.m_nRotateBegin,363);
			Axis_XZ.XZ_AxisCmd.AxisPara.rAbsVelocity:=XZ_Velocity;
			
			IF WorkStation_TCP.PLC_RECV1.m_nSocketType=1 THEN
				Axis_XZ.XZ_AxisCmd.bAbs:=TRUE;
			END_IF;
			
			(*4.到位后2秒跳转*)
			IF ABS(Axis_XZ.XZ_AxisState.rActPosition-WorkStation_TCP.PLC_RECV1.m_nRotateBegin)<1 AND Axis_XZ.XZ_AxisState.bStandStill THEN
				Step_CBCT:=220;	
			END_IF
		
		220://中间状态清零
			Axis_XZ.XZ_AxisCmd.bAbs:=FALSE;
			Axis_QJ.QJ_AxisCmd.bAbs:=FALSE;
			Step_CBCT:=230;
			
		230://用户按7键，床自动走到预设位置
			(*1.按7键关闭7灯*)
			IF CTBOX_RS232.CTBOX_KEY_Manual THEN
				LampCmd7:=E_LampCmd.关闭;
				WorkStation_TCP.PLC_SEND1.m_nFocus:=0;	//关闭按键提示0228
			END_IF
			
			(*2.触发床运动*)
			R_TRIG_G2(CLK:=CTBOX_RS232.CTBOX_KEY_Manual , Q=> );
			Axis_QJ.QJ_AxisCmd.AxisPara.rAbsPosition:=LIMIT(0,WorkStation_TCP.PLC_RECV1.m_fScanTop,900);
			Axis_QJ.QJ_AxisCmd.bAbs:=R_TRIG_G2.Q;
			
			(*3.跳转指令*)
			IF ABS(Axis_QJ.QJ_AxisState.rActPosition-WorkStation_TCP.PLC_RECV1.m_fScanTop)<1 AND (LampCmd7=E_LampCmd.关闭) THEN //保证必须按下7键
				WorkStation_TCP.PLC_SEND1.m_nMoveState:=1; //send [9]	//0-准备过程中 1-准备完成 2-曝光中 3-本次扫描结束
			ELSE
				WorkStation_TCP.PLC_SEND1.m_nMoveState:=0; //send [9]	//0-准备过程中 1-准备完成 2-曝光中 3-本次扫描结束
			END_IF
			
			(*4.延迟跳转，保证send [9]发送*)
			TON_CT_G[11](IN:=(WorkStation_TCP.PLC_SEND1.m_nMoveState=1) , PT:=T#1100MS , Q=> , ET=> );
			IF TON_CT_G[11].Q THEN
				Step_CBCT:=60;
			END_IF
	END_CASE
END_ACTION

ACTION _a_Homing_active:

(*回零*)

		TON_Home(IN:= TRUE, PT:= T#10S, Q=> , ET=> );

		Axis_XZ.XZ_AxisCmd.AxisPara.rSetPosition:=GVL_Retain.rXZ_Position;
		Axis_XZ.XZ_AxisCmd.bSetPos:=TON_Home.Q;//赋值为true
	
		Axis_QJ.QJ_AxisCmd.AxisPara.rSetPosition:=GVL_Retain.rQJ_Position;
		Axis_QJ.QJ_AxisCmd.bSetPos:=TON_Home.Q;
		
		
	(*5.2 执行回零命令*)
	
		LampCmd5:=E_LampCmd.关闭;
		LampCmd6:=E_LampCmd.关闭;
		LampCmd7:=E_LampCmd.关闭;
		LampCmd8:=E_LampCmd.关闭;
	
		IF (Axis_QJ.fbMC_SetPostiong.Done AND Axis_XZ.fbMC_SetPostiong.Done) THEN
			bHomingDone:=TRUE;
			Step_Home:=10;
		ELSE
			bHomingDone:=FALSE;	
		END_IF
END_ACTION

ACTION _a_Emergercy_entry_1:

GVL_State.iPLC_State:=330;
END_ACTION

ACTION _a_QuickCT_exit:


	LampCmd5:=E_LampCmd.关闭;
	LampCmd6:=E_LampCmd.关闭;
	LampCmd7:=E_LampCmd.关闭;
	LampCmd8:=E_LampCmd.关闭;
	
	Entity_IO.bTriggerOut:=FALSE;
END_ACTION

TRANSITION T_StandardCT:

(*进入旋转轴运动模式*)
	WorkStation_TCP.PLC_RECV1.m_nSocketType=1 AND WorkStation_TCP.PLC_RECV1.m_nExpId=3
END_TRANSITION

ACTION _a_SelfCheck_entry:

//	Axis_XZ.XZ_AxisCmd.bPower:=TRUE;//上使能
//	Axis_QJ.QJ_AxisCmd.bPower:=TRUE;//上使能
	
	Axis_XZ.XZ_AxisCmd.bPower:=FALSE;//上使能
	Axis_QJ.QJ_AxisCmd.bPower:=FALSE;//上使能
END_ACTION

ACTION AirHigh_entry:


Step_Air:=0; 

GVL_State.iPLC_State:=350;//空气校正


Entity_io.bXraySwitch:=TRUE;//PF CLK信号切换继电器 不得电是默认BUCKY触发
END_ACTION

TRANSITION T_HighDefinCT:


(*进入CBCT扫描*)
	WorkStation_TCP.PLC_RECV1.m_nSocketType=1 AND (WorkStation_TCP.PLC_RECV1.m_nExpId=5 OR WorkStation_TCP.PLC_RECV1.m_nExpId=3)
END_TRANSITION

ACTION _a_DynamicsDR_exit:

	Entity_IO.bTriggerOut:=FALSE;
	Entity_IO.bXaryOne:=FALSE;
	Entity_IO.bXaryTwo:=FALSE;
END_ACTION

ACTION _a_Init_active_1:



			(*1.给上位机发送的数据*)
			WorkStation_TCP.PLC_SEND1.m_nMoveState:=0;			//send[9]
			Axis_XZ.XZ_AxisCmd.bAbs:=FALSE;
			bScoutLast := FALSE;
			
			(*2.运动准备数据*)
			(*2.1 写入旋转速度参数*)
			Axis_XZ.XZ_AxisCmd.AxisPara.rAbsVelocity:=36;//定位像扫描按照设定速度运动
			
(*
			TON_S30(IN:= FALSE );
			TON_S40(IN:= FALSE);TON_S50(IN:= FALSE);
			TON_S70(IN:= FALSE);TON_S80(IN:= FALSE);
			TOF_S50(IN:= FALSE);TON_S60(IN:= FALSE);
			TON_S52(IN:= FALSE );TON_S41(IN:=FALSE);
			TON_S43(IN:= FALSE );TON_S20_ABS(IN:=FALSE);
			Axis_XZ.XZ_AxisCmd.bAbs:=FALSE;
*)
END_ACTION

ACTION _a_ShutDown_active_1:

(*关机模式*)

(*1.伺服电机下使能*)
	Axis_XZ.XZ_AxisCmd.bPower:=FALSE;
	Axis_QJ.QJ_AxisCmd.bPower:=FALSE;
		
(*2.运动都停止*)
	Axis_XZ.XZ_AxisCmd.bStop:=FALSE;
	Axis_QJ.QJ_AxisCmd.bStop:=FALSE;
	Motor_SJ(Enable:= FALSE);

(*3.无法出束，控制二档信号*)
	Entity_IO.bXaryTwo:=FALSE;
	Entity_IO.bXaryOne:=FALSE;
	Entity_IO.bXaryFlu:=FALSE;
	
(*4.记录参数*)

(*处理旋转电机度数问题*)
(*	IF Axis_XZ.XZ_AxisState.rActPosition<355 THEN
		Axis_XZ.XZ_AxisCmd.bPower	:=FALSE;
		Axis_XZ.XZ_AxisCmd.bStop	:=FALSE;
		bOver:=TRUE;
	ELSE
		CASE Step_ShutDown OF 
		0:
			Axis_XZ.XZ_AxisCmd.AxisPara.rAbsPosition:=350;	//相对位移
			Axis_XZ.XZ_AxisCmd.AxisPara.rAbsVelocity:=10; 	//相对速度
			Step_ShutDown:=10;
		
		10:
			Axis_XZ.XZ_AxisCmd.bAbs:=TRUE;
			IF ABS(Axis_XZ.XZ_AxisState.rActPosition-350)<1 AND Axis_XZ.XZ_AxisState.bStandStill THEN
				Step_ShutDown:=20;
			END_IF
			
		20:
			Axis_XZ.XZ_AxisCmd.bRel:=FALSE;
			bOver:=TRUE;
		END_CASE;
	END_IF
*)
END_ACTION

ACTION _a_DynamicsDR_active:


	CASE Step_DynamicDR OF 
		0:	//初始化准备流程
			(*1.给上位机发送的数据*)
			WorkStation_TCP.PLC_SEND1.m_nMoveState:=0;			//send[9]
			
			(*2.运动准备数据*)
			(*2.1 写入旋转速度参数*)
			Axis_XZ.XZ_AxisCmd.AxisPara.rAbsVelocity:=36;//定位像扫描按照设定速度运动
			Axis_XZ.XZ_AxisCmd.bAbs		:=FALSE;
			bStaticDRLast 				:=FALSE;
			
			(*3.//运动过程中变量复位标志*)
			FOR i:=1 TO 50 BY 1 DO 
				TON_DR_S[i](IN:= FALSE);
			END_FOR
		
			(*4.跳转*)
			Step_DynamicDR:=10;

		10://开启运动
			(*1.给上位机发送的数据*)
			WorkStation_TCP.PLC_SEND1.m_nExpStates	:=1;//为曝光状态，枚举值，0:idle（空闲） 1:prep（训机） 2: ready（训机结束，准备完成，可以出束） 3: XrayOn（出射线） 4:XrayOff（关射线） 5 error；
			WorkStation_TCP.PLC_SEND1.m_nMoveState	:=0;//起始、终止状态， 默认值-1， 0为当前扫描方案（与常规意义不同，注意区别）处于准备好状态，可以准备扫描；1为当前扫描方案结束，运动过程中值为-1
			WorkStation_TCP.PLC_SEND1.m_nScanProType:=2;//执行扫描方案的类型，0为自动扫描，1为手动扫描，2为无设置意义的值，默认值为2
	
			(*2.旋转轴运动*)
			TON_DR_S[1](IN:= TRUE, PT:=T#500MS);
			Axis_XZ.XZ_AxisCmd.bAbs:=TON_DR_S[1].Q;
			Axis_XZ.XZ_AxisCmd.AxisPara.rAbsPosition:=LIMIT(-4,WorkStation_TCP.PLC_RECV1.m_nRotateBegin,363);

			(*3.跳转下一个步骤*)	
			IF  ABS(Axis_XZ.XZ_AxisState.rActPosition-WorkStation_TCP.PLC_RECV1.m_nRotateBegin)<=1 AND Axis_XZ.XZ_AxisState.bStandStill THEN
				Step_DynamicDR:=20;
			END_IF
			
		20:
			IF DT_Xray.DR_Para=66 THEN 			//DR模式下写参完成
				Step_StaticDR:=30;
			END_IF
			
		30://按下1档，或踩下脚闸信号后，输出信号给射线源
			(*1.一二档信号输出处理*)
			IF Entity_IO.bXrayOneInput OR Entity_IO.bXayExpoInput OR Entity_IO.bXrayFluInput THEN	//一档信号，或脚咋信号
				Entity_IO.bXaryOne:=TRUE;
			ELSE
				Entity_IO.bXaryOne:=FALSE;
			END_IF
			
			IF Entity_IO.bXaryOne AND Entity_IO.bXrayFluInput THEN
				Entity_IO.bXaryTwo:=TRUE;
			END_IF
			
			(*3.写射线源参数及跳转处理*)
			IF Entity_IO.bXaryTwo AND DT_Xray.DR_Para=66 THEN 			//DR模式下写参完成
				Step_DynamicDR:=40;
			END_IF
			TimeDRExpS:=LIMIT(T#1MS,REAL_TO_TIME(WorkStation_TCP.PLC_RECV1.m_nMS/10),T#30S);			//获取上位机发送的曝光时间//这里有个最大时间
			
			(*4.发送给上位机的数据*)
			WorkStation_TCP.PLC_SEND1.m_nMoveState	:=0;//起始、终止状态， 默认值-1， 0为当前扫描方案（与常规意义不同，注意区别）处于准备好状态，可以准备扫描；1为当前扫描方案结束，运动过程中值为-1
		
		40://PLC延迟射线源曝光时间后，触发探测器采一张图
			WorkStation_TCP.PLC_SEND1.m_nExpStates	:=1;//为曝光状态，枚举值，0:idle（空闲） 1:prep（训机） 2: ready（训机结束，准备完成，可以出束） 3: XrayOn（出射线） 4:XrayOff（关射线） 5 error；
			TON_DR_S[2](IN:= TRUE, PT:=TimeDRExpS+T#30MS);		//内触发06模式出图采集
			IF TON_DR_S[2].Q THEN
				Step_DynamicDR:=50;
			END_IF;
			
		50://跳出扫描
			GVL_SCAN.bJumpScan:=TRUE;
	END_CASE
	
	
(*		
		20://开启Pannel和CTBox运动感权限
			(*2.1 升降轴运动*)
			Motor_SJ(Enable:= TRUE);
			
			(*2.2 前进轴控制*)
			(*2.1 相对运动*)
			(*2.1 旋转轴一键运动到0°运动*)
			Axis_XZ.XZ_AxisCmd.AxisPara.rAbsPosition:=0;//目标位置
			Axis_XZ.XZ_AxisCmd.AxisPara.rAbsVelocity:=36;//运动速度36
			Axis_XZ.XZ_AxisCmd.bAbs:=Entity_IO.LeftPannel_DistanceMove OR Entity_IO.RightPannel_DistanceMove;
			
			(*2.2 点动和绝对运动合并程序*)
			Axis_QJ.QJ_AxisCmd.AxisPara.rAbsVelocity:=80;
			(*2.2.1 点动触发逻辑*)
			R_TRIG_Jog(CLK:= (Entity_IO.LeftPannel_BedFore OR Entity_IO.RightPannel_BedFore OR CTBOX_RS232.CTBOX_KEY_BedFore)
						OR (Entity_IO.LeftPannel_BedBack OR Entity_IO.RightPannel_BedBack OR CTBOX_RS232.CTBOX_KEY_BedBack), Q=> ); //获取上升沿
			F_TRIG_Jog(CLK:= (Entity_IO.LeftPannel_BedFore OR Entity_IO.RightPannel_BedFore OR CTBOX_RS232.CTBOX_KEY_BedFore)
						OR (Entity_IO.LeftPannel_BedBack OR Entity_IO.RightPannel_BedBack OR CTBOX_RS232.CTBOX_KEY_BedBack), Q=> ); //获取上升沿
	
			(*2.2.2 点动最大最小位置，绝对运动走记录值*)
			IF Entity_IO.LeftPannel_BedFore OR Entity_IO.RightPannel_BedFore OR CTBOX_RS232.CTBOX_KEY_BedFore THEN
				Axis_QJ.QJ_AxisCmd.AxisPara.rAbsPosition:=900;
			ELSE
				IF Entity_IO.LeftPannel_BedBack OR Entity_IO.RightPannel_BedBack OR CTBOX_RS232.CTBOX_KEY_BedBack THEN
					Axis_QJ.QJ_AxisCmd.AxisPara.rAbsPosition:=0;
				ELSE
					Axis_QJ.QJ_AxisCmd.AxisPara.rAbsPosition:=LIMIT(0,GVL_Retain.rBedRecordLength,900); 
				END_IF
			END_IF
			
			(*2.2.3 触发绝对运动，按键或者触发走记录位置*)
			Axis_QJ.QJ_AxisCmd.bAbs	:=R_TRIG_Jog.Q OR  Entity_IO.LeftPannel_MoveRecordPos OR Entity_IO.RightPannel_MoveRecordPos;
			
			(*2.2.4 触发停止*)
			R_RelStop(CLK:= (Axis_QJ.QJ_AxisState.rActPosition>901), Q=> ); 
			Axis_QJ.QJ_AxisCmd.bStop:=F_TRIG_Jog.Q OR R_RelStop.Q;
			
			IF Entity_IO.bXrayOneInput OR Entity_IO.bXayExpoInput OR Entity_IO.bXrayFluInput THEN 	//一档信号，或脚咋信号
				Step_DynamicDR:=30;
			END_IF
*)
END_ACTION

ACTION _a_Wait_active:

TON_Power(IN:=TRUE,PT:=T#13S);
END_ACTION

ACTION _a_Idle_active:

(*待机工作状态*)
	
	CASE Step_Idle OF
	0: //中间状态复位
		Entity_IO.bXaryOne:=FALSE;				//试一试在这里高压会不会报错
		Entity_IO.bXaryTwo:=FALSE;				//试一试在这里高压会不会报错
		Entity_IO.bXaryFlu:=FALSE;	
		WorkStation_TCP.PLC_SEND1.m_nFocus:=0;	//按键提示清零0228
		TON_I00(IN:=FALSE , PT:= , Q=> , ET=> );
		TON_I10(IN:=FALSE , PT:= , Q=> , ET=> );
		TON_I20(IN:=FALSE , PT:= , Q=> , ET=> );
		TON_I30(IN:=FALSE , PT:= , Q=> , ET=> );
		TON_I40(IN:=FALSE , PT:= , Q=> , ET=> );
		TON_I50(IN:=FALSE , PT:= , Q=> , ET=> );
		TON_IDLE(IN:=FALSE, PT:= , Q=> , ET=> );
		Step_Idle:=10;
		
	10:	//所有运动立刻停止，所有灯关闭
		TON_I00(IN:=TRUE , PT:=T#1S , Q=> , ET=> );
		TON_I10(IN:=TRUE , PT:=T#1S , Q=> , ET=> );
		Axis_QJ.QJ_AxisCmd.bStop:=TON_I00.Q;
		Axis_XZ.XZ_AxisCmd.bStop:=TON_I10.Q;
		
		LampCmd5:=E_LampCmd.关闭;
		LampCmd6:=E_LampCmd.关闭;
		LampCmd7:=E_LampCmd.关闭;
		LampCmd8:=E_LampCmd.关闭;
		
		TON_IDLE(IN:= TRUE, PT:=T#2S , Q=> , ET=> );
		IF TON_IDLE.Q THEN
			Step_Idle:=20;
		END_IF
		
	20:	//中间变量复位
		Axis_QJ.QJ_AxisCmd.bStop:=FALSE;
		Axis_XZ.XZ_AxisCmd.bStop:=FALSE;
		TON_IDLE(IN:= FALSE, PT:=T#2S , Q=> , ET=> );
		Step_Idle:=30;
		
	30:	//待机模式准备，开启点动运动权限
		GVL_State.iPLC_State:=40;
		
		(*1.给上位机发送数据*)
		WorkStation_TCP.PLC_SEND1.m_nExpStates	:=1;//[4]为曝光状态，枚举值，0:idle（空闲） 1:prep（训机） 2: ready（训机结束，准备完成，可以出束） 3: XrayOn（出射线） 4:XrayOff（关射线） 5 error；
		WorkStation_TCP.PLC_SEND1.m_nMoveState	:=0;//[9]起始、终止状态， 默认值-1， 0为当前扫描方案处于准备好状态，可以准备扫描；1为当前扫描方案结束，运动过程中值为-1
		WorkStation_TCP.PLC_SEND1.m_nScanProType:=2;//[16]执行扫描方案的类型，0为自动扫描，1为手动扫描，2为无设置意义的值，默认值为2
		
		(*2.开启前进轴和升降轴运动*)
		(*2.1 升降轴运动*)
		Motor_SJ(Enable:= TRUE);
		
		(*2.2 前进轴控制*)
		(*2.1 旋转轴一键运动到0°运动*)
		Axis_XZ.XZ_AxisCmd.AxisPara.rAbsPosition:=0;//目标位置
		Axis_XZ.XZ_AxisCmd.AxisPara.rAbsVelocity:=36;//运动速度36
		Axis_XZ.XZ_AxisCmd.bAbs:=Entity_IO.LeftPannel_DistanceMove OR Entity_IO.RightPannel_DistanceMove;
		
		(*2.2 点动和绝对运动合并程序*)
		Axis_QJ.QJ_AxisCmd.AxisPara.rAbsVelocity:=80;
		(*2.2.1 点动触发逻辑*)
		R_TRIG_Jog(CLK:= (Entity_IO.LeftPannel_BedFore OR Entity_IO.RightPannel_BedFore OR CTBOX_RS232.CTBOX_KEY_BedFore), Q=> ) ; //获取上升沿
		R_TRIG_Jog1(CLK:= (Entity_IO.LeftPannel_BedBack OR Entity_IO.RightPannel_BedBack OR CTBOX_RS232.CTBOX_KEY_BedBack) , Q=> ) ; //获取上升沿
		
		F_TRIG_Jog(CLK:= (Entity_IO.LeftPannel_BedFore OR Entity_IO.RightPannel_BedFore OR CTBOX_RS232.CTBOX_KEY_BedFore), Q=> ); //获取下降沿
		F_TRIG_Jog1(CLK:=(Entity_IO.LeftPannel_BedBack OR Entity_IO.RightPannel_BedBack OR CTBOX_RS232.CTBOX_KEY_BedBack) , Q=> ); //获取下降沿

		(*2.2.2 点动最大最小位置，绝对运动走记录值*)
		IF Entity_IO.LeftPannel_BedFore OR Entity_IO.RightPannel_BedFore OR CTBOX_RS232.CTBOX_KEY_BedFore THEN
			Axis_QJ.QJ_AxisCmd.AxisPara.rAbsPosition:=900;
		ELSE
			IF Entity_IO.LeftPannel_BedBack OR Entity_IO.RightPannel_BedBack OR CTBOX_RS232.CTBOX_KEY_BedBack THEN
				Axis_QJ.QJ_AxisCmd.AxisPara.rAbsPosition:=0;
			ELSE
				Axis_QJ.QJ_AxisCmd.AxisPara.rAbsPosition:=LIMIT(0,GVL_Retain.rBedRecordLength,900); 
			END_IF
		END_IF
		
		(*2.2.3 触发绝对运动，按键或者触发走记录位置*)
		Axis_QJ.QJ_AxisCmd.bAbs	:=(R_TRIG_Jog.Q OR R_TRIG_Jog1.Q OR  Entity_IO.LeftPannel_MoveRecordPos OR Entity_IO.RightPannel_MoveRecordPos) AND Axis_QJ.QJ_AxisState.bStandStill;
		
		(*2.2.4 触发停止*)
		R_RelStop(CLK:= (Axis_QJ.QJ_AxisState.rActPosition>901), Q=> ); 
		Axis_QJ.QJ_AxisCmd.bStop:=F_TRIG_Jog.Q OR F_TRIG_Jog1.Q  OR R_RelStop.Q;
		
	END_CASE
	
	
(*		Axis_QJ.QJ_AxisCmd.AxisPara.rRelVelocity:=80;
		Axis_QJ.QJ_AxisCmd.AxisPara.rRelPosition:=50;
		IF Axis_QJ.QJ_AxisState.rActPosition<=900 THEN
			Axis_QJ.QJ_AxisCmd.bRel:=Entity_IO.LeftPannel_DistanceMove OR Entity_IO.RightPannel_DistanceMove;
		ELSE
			Axis_QJ.QJ_AxisCmd.bRel:=FALSE;
		END_IF
*)
END_ACTION

ACTION _a_Error_exit:


		Axis_QJ.QJ_AxisCmd.bReset:=FALSE;
		Axis_XZ.XZ_AxisCmd.bReset:=FALSE;
END_ACTION

ACTION _a_HighDefinCT_exit:

	LampCmd5:=E_LampCmd.关闭;
	LampCmd6:=E_LampCmd.关闭;
	LampCmd7:=E_LampCmd.关闭;
	LampCmd8:=E_LampCmd.关闭;
	
	Entity_IO.bTriggerOut:=FALSE;
	iActNumPulse:=0;
	
	Entity_io.bXraySwitch:=FALSE;//PF CLK信号切换继电器 不得电是默认BUCKY触发
END_ACTION

ACTION _a_Homing_entry:

	GVL_State.iPLC_State:=30;
	Step_Home:=0;
	
	Axis_QJ.QJ_AxisCmd.bSetHomePara:=FALSE;
	Axis_XZ.XZ_AxisCmd.bSetHomePara:=FALSE;
	
	bHomingDone:=FALSE;
	
	Axis_XZ.XZ_AxisCmd.bHome:=FALSE;
	Axis_QJ.QJ_AxisCmd.bHome:=FALSE;
	
	TON_Home(IN:= FALSE);
	
	Axis_XZ.XZ_AxisCmd.bPower:=TRUE;
	Axis_QJ.QJ_AxisCmd.bPower:=TRUE;
END_ACTION

ACTION _a_Debug_entry:


GVL_State.iPLC_State:=320;
END_ACTION

ACTION _a_Init_active:

TON_Power(IN:=FALSE);
InitMotor(); //电机初始化程序
END_ACTION

ACTION _a_Logic_active:


Entity_IO();
CTBOX_RS232();
WorkStation_TCP();
WorkMode();
//Trigger_HaoboPannel();

(*1.激光灯控制*)
(*按键后30秒自动停止输出，如果在30秒之内再次按键，下降沿有效，则立刻停止输出*)
	IF WorkMode.iWorkMode=99 THEN
		Entity_IO.bLaserOut:=bDebug_Laser;
	ELSE
		TP_Laser(IN:=Entity_IO.LeftPannel_LaserButton OR Entity_IO.RightPannel_LaserButton , PT:=T#5MS , Q=> , ET=> );
		R_TRIG1(CLK:=TP_Laser.Q , Q=> );
		TOF_Laser(IN:=TP_Laser.Q , PT:=T#60S , Q=> , ET=>TOF_ET );
		IF TOF_Laser.Q THEN
			IF R_TRIG1.Q THEN
				IF Entity_IO.bLaserOut THEN
					Entity_IO.bLaserOut:= FALSE;
				ELSE
					Entity_IO.bLaserOut:= TRUE;
				END_IF
			END_IF
		ELSE
			Entity_IO.bLaserOut:= FALSE;
		END_IF
	
		Entity_IO.bLeftPannel_LED2:=Entity_IO.bLaserOut;
		Entity_IO.bRightPannel_LED1:=Entity_IO.bLaserOut;
	END_IF

(*2.延迟断电功能*)
	TOF_PowerDelayMax(IN:= 	Entity_IO.bKeySwitch , 			PT:= T#15S, 	Q=> );				//无论什么错误 15秒都关机
	TOF_PowerDelay(IN:= 	Entity_IO.bKeySwitch AND bOver, PT:= T#5S,	 	Q=> );				//关机流程结束后
	Entity_IO.bDelayPower:= TOF_PowerDelayMax.Q OR TOF_PowerDelay.Q;
	
(*3.射线源1和2档对应输出功能及黄色射线指示灯功能*)

	IF (Entity_IO.bXaryTwo OR Entity_IO.bXaryFlu) AND Entity_IO.bDoorLock THEN 		//门已关闭的情况下
		Entity_IO.bLightYellow:=TRUE;
	ELSE
		Entity_IO.bLightYellow:=FALSE;
	END_IF

(*4.中止扫描*)
	TON_StopScan(IN:= CTBOX_RS232.CTBOX_KEY_Stop, PT:= T#1S, Q=> , ET=> );
	
(*5.记录预设位置操作*)
	IF Entity_IO.LeftPannel_RecordPos OR Entity_IO.RightPannel_RecordPos THEN
		GVL_Retain.rBedRecordHeight:=Entity_IO.rRealPos;
		GVL_Retain.rBedRecordLength:=LREAL_TO_REAL(Axis_QJ.QJ_AxisState.rActPosition);
	ELSE
		GVL_Retain.rBedRecordHeight:=GVL_Retain.rBedRecordHeight;
		GVL_Retain.rBedRecordLength:=GVL_Retain.rBedRecordLength;
	END_IF
	
(*6.日志记录*)
	RecordLog();

(*7.旋转轴零位写入*)
	IF bSetXZ_Zero THEN
		GVL_Retain.rXZ_Zero:=rSetXZ_Zero;
	END_IF

(*8.旋转轴和前进轴断电保持当前位置，用做设置当前位置用*)
	IF  GVL_State.iPLC_State> 30 THEN
		GVL_Retain.rXZ_Position:=AXIS_XZ.XZ_AxisState.rActPosition;
		GVL_Retain.rQJ_Position:=AXIS_QJ.QJ_AxisState.rActPosition;
	END_IF



//记录曝光时间，快速扫描模式，测试用		
(*	IF GVL_State.iPLC_State=240 THEN
		
		R_TRIG_SS(CLK:= Entity_IO.bXrayExp, Q=> );	
		F_TRIG_SS(CLK:= Entity_IO.bXrayExp, Q=> );
		
		IF R_TRIG_SS.Q THEN
			Second1:=LS_ReadDintDT_1.uiSecond;
			Minute1:=LS_ReadDintDT_1.uiMinute;
		END_IF;
		
		IF F_TRIG_SS.Q THEN
			Second2:=LS_ReadDintDT_1.uiSecond;
			Minute2:=LS_ReadDintDT_1.uiMinute;
		END_IF; 
	END_IF
*)
END_ACTION

ACTION _a_Wait_exit:
GVL_State.iPLC_State:=10;
END_ACTION

ACTION _a_StaticDR_active:


	CASE Step_StaticDR OF 
		0:	//初始化准备流程
			(*1.给上位机发送的数据*)
			WorkStation_TCP.PLC_SEND1.m_nMoveState:=0;			//send[9]
			WorkStation_TCP.PLC_SEND1.m_nFocus:=0;	
			
			(*2.运动准备数据*)
			(*2.1 写入旋转速度参数*)
			Axis_XZ.XZ_AxisCmd.AxisPara.rAbsVelocity:=36;//定位像扫描按照设定速度运动
			Axis_XZ.XZ_AxisCmd.bAbs		:=FALSE;
			bStaticDRLast 				:=FALSE;
			
			(*3.//运动过程中变量复位标志*)
			FOR i:=1 TO 50 BY 1 DO 
				TON_DR_S[i](IN:= FALSE);
			END_FOR
			Entity_IO.bXaryTwo:=FALSE;Entity_IO.bXaryOne:=FALSE;
			
			F_TRIG_S1(CLK:=FALSE);
			
			(*4.跳转*)
			Step_StaticDR:=10;

		10://开启运动
			(*1.给上位机发送的数据*)
			WorkStation_TCP.PLC_SEND1.m_nExpStates	:=1;//为曝光状态，枚举值，0:idle（空闲） 1:prep（训机） 2: ready（训机结束，准备完成，可以出束） 3: XrayOn（出射线） 4:XrayOff（关射线） 5 error；
			WorkStation_TCP.PLC_SEND1.m_nMoveState	:=0;//起始、终止状态， 默认值-1， 0为当前扫描方案（与常规意义不同，注意区别）处于准备好状态，可以准备扫描；1为当前扫描方案结束，运动过程中值为-1
			WorkStation_TCP.PLC_SEND1.m_nScanProType:=2;//执行扫描方案的类型，0为自动扫描，1为手动扫描，2为无设置意义的值，默认值为2
	
			(*2.旋转轴运动*)
			TON_DR_S[1](IN:= TRUE, PT:=T#500MS);
			Axis_XZ.XZ_AxisCmd.bAbs:=TON_DR_S[1].Q;
			Axis_XZ.XZ_AxisCmd.AxisPara.rAbsPosition:=LIMIT(-4,WorkStation_TCP.PLC_RECV1.m_nRotateBegin,363);

			(*3.跳转下一个步骤*)	
			IF  ABS(Axis_XZ.XZ_AxisState.rActPosition-WorkStation_TCP.PLC_RECV1.m_nRotateBegin)<=1 AND Axis_XZ.XZ_AxisState.bStandStill THEN(**)
				Step_StaticDR:=20;
			END_IF
			
		20:
			TON_DR_S[10](IN:=FALSE);
			TON_DR_S[5](IN:= TRUE, PT:=T#1S);
			 bXrayOneDR:=FALSE;
			WorkStation_TCP.PLC_SEND1.m_nFocus:=1;	
			IF DT_Xray.DR_Para=66 AND TON_DR_S[5].Q THEN 			//DR模式下写参完成
				Step_StaticDR:=30;
			END_IF
			
		30://按下1档，或踩下脚闸信号后，输出信号给射线源
			(*1.一二档信号输出处理*)
			TOF_DR111(IN:=(Entity_IO.bXrayOneInput OR Entity_IO.bXayExpoInput) , PT:= T#2S, Q=> Entity_IO.bXaryOne, ET=> );
			TOF_DR22(IN:=(Entity_IO.bXrayTwoInput OR Entity_IO.bXayExpoInput) , PT:= T#2S, Q=> Entity_IO.bXaryTwo, ET=> );
			
			(*2.判断是否最后一次扫描标志位*)
			IF WorkStation_TCP.PLC_RECV1.m_nLastMsg=1 THEN bStaticDRLast := TRUE;
			ELSE bStaticDRLast := FALSE;
			END_IF
			
			(*3.写射线源参数及跳转处理*)
			IF Entity_IO.bXaryTwo THEN
				Step_StaticDR:=35;
			END_IF
			
			TimeDRExpS:=LIMIT(T#1MS,REAL_TO_TIME(WorkStation_TCP.PLC_RECV1.m_nMS),T#15S);			//获取上位机发送的曝光时间
			
			(*4.发送给上位机的数据*)
			WorkStation_TCP.PLC_SEND1.m_nMoveState	:=0;//起始、终止状态， 默认值-1， 0为当前扫描方案（与常规意义不同，注意区别）处于准备好状态，可以准备扫描；1为当前扫描方案结束，运动过程中值为-1
		
			IF TOF_DR111.Q THEN
				WorkStation_TCP.PLC_SEND1.m_nFocus:=0;					//按键关闭
			ELSE
				WorkStation_TCP.PLC_SEND1.m_nFocus:=1;					//按键提示
			END_IF
			
			(*5.二挡信号刚给就出一张图*)
			R_Static_Tigger(CLK:= Entity_IO.bXaryTwo, Q=>Entity_IO.bTriggerOut );
			
			(*6 按了1档，又松了，跳到待机模式*)
			 F_DR_Jump(CLK:= TOF_DR111.Q, Q=> );	//1114
			 R_DR_Jump(CLK:= Entity_IO.bXaryOne, Q=> );
			 IF R_DR_Jump.Q THEN
				 bXrayOneDR:=TRUE;
			 END_IF
			 
			 IF bXrayOneDR AND F_DR_Jump.Q AND NOT(Entity_IO.bXaryTwo) THEN
				 GVL_SCAN.bJumpScan:=TRUE;
			 END_IF
			
		35:
			TOF_DR22(IN:=(Entity_IO.bXrayTwoInput OR Entity_IO.bXayExpoInput) , PT:= T#4S, Q=> Entity_IO.bXaryTwo, ET=> );
			R_Static_Tigger(CLK:= FALSE);
			Entity_IO.bTriggerOut:=FALSE;
			WorkStation_TCP.PLC_SEND1.m_nFocus:=0;					//按键关闭
			TON_DR_S[4](IN:=TRUE , PT:=T#3S , Q=> , ET=> );
		
			IF TON_DR_S[4].Q AND Entity_IO.bXaryTwo THEN
				Step_StaticDR:=40;
			END_IF
		
		40://PLC延迟射线源曝光时间后，触发探测器采一张图
			TOF_DR22(IN:=(Entity_IO.bXrayTwoInput OR Entity_IO.bXayExpoInput) , PT:= T#1S, Q=> Entity_IO.bXaryTwo, ET=> );
			F_TRIG_S1(CLK:= Entity_IO.bXaryTwo, Q=> );
			
			WorkStation_TCP.PLC_SEND1.m_nExpStates	:=1;//为曝光状态，枚举值，0:idle（空闲） 1:prep（训机） 2: ready（训机结束，准备完成，可以出束） 3: XrayOn（出射线） 4:XrayOff（关射线） 5 error；
			TON_DR_S[2](IN:= TRUE, PT:=TimeDRExpS);
			Entity_IO.bTriggerOut:=TON_DR_S[2].Q;	//或二挡信号消失，立刻触发一次采图
			
			IF TON_DR_S[2].Q OR F_TRIG_S1.Q THEN
				Step_StaticDR:=45;
			END_IF

		45:		
			Entity_IO.bXaryOne:=FALSE;
			Entity_IO.bXaryTwo:=FALSE;
			Entity_IO.bTriggerOut:=FALSE;
			TOF_DR111(IN:=FALSE);TOF_DR22(IN:=FALSE);
			
			TON_DR_S[10](IN:=TRUE , PT:=T#1500MS , Q=> , ET=> );
			IF TON_DR_S[10].Q THEN
				Step_StaticDR:=50;
			END_IF
			
		50://判断是否最后一次扫描
			(*1.给上位机发送的数据*)
			WorkStation_TCP.PLC_SEND1.m_nMoveState:=3; //send [9]
			
			(*2.判断是否最后一次扫描*)
			TON_DR_S[3](IN:=TRUE , PT:=T#1S , Q=> , ET=> );
			IF TON_DR_S[3].Q THEN
				IF (WorkStation_TCP.PLC_RECV1.m_nCircleIndex+1)>=(WorkStation_TCP.PLC_RECV1.m_nCircleCount) AND bStaticDRLast  THEN//最后一次扫描退出
					GVL_SCAN.bJumpScan:=TRUE;
				END_IF
			END_IF
		
			(*3.不是最后一次增加跳转判断增加跳转接着扫*)
			IF WorkStation_TCP.PLC_RECV1.m_nSocketType=1 THEN 	//增加第二次运动判断，m_nSocketType=1 
				Step_StaticDR:=00;
			END_IF
	END_CASE
	
	
(*			
			TON_DR_S[22](IN:= TRUE, PT:=T#10M);
			TON_DR_S[23](IN:= TRUE, PT:=T#900MS);
			IF TON_DR_S[23].Q=FALSE THEN
				Blink_StaticDR_Temp(ENABLE:= TON_DR_S[2].Q, TIMELOW:=T#100MS , TIMEHIGH:= T#100MS, OUT=>Entity_IO.bTriggerOut );
			ELSE
				Entity_IO.bTriggerOut:=TON_DR_S[22].Q;
			END_IF;
			
			IF TON_DR_S[22].Q THEN
				Step_StaticDR:=45;
			END_IF
			
			IF TON_DR_S[2].Q THEN
				Entity_IO.bXaryOne:=FALSE;
				Entity_IO.bXaryTwo:=FALSE;
			END_IF;
*)			
	
	(*	20://开启Pannel和CTBox运动感权限
			(*2.1 升降轴运动*)
			Motor_SJ(Enable:= TRUE);
			
			(*2.2 前进轴控制*)
			(*2.1 旋转轴一键运动到0°运动*)
			Axis_XZ.XZ_AxisCmd.AxisPara.rAbsPosition:=0;//目标位置
			Axis_XZ.XZ_AxisCmd.AxisPara.rAbsVelocity:=36;//运动速度36
			Axis_XZ.XZ_AxisCmd.bAbs:=Entity_IO.LeftPannel_DistanceMove OR Entity_IO.RightPannel_DistanceMove;
			
			(*2.2 点动和绝对运动合并程序*)
			Axis_QJ.QJ_AxisCmd.AxisPara.rAbsVelocity:=80;
			(*2.2.1 点动触发逻辑*)
			R_TRIG_Jog(CLK:= (Entity_IO.LeftPannel_BedFore OR Entity_IO.RightPannel_BedFore OR CTBOX_RS232.CTBOX_KEY_BedFore)
						OR (Entity_IO.LeftPannel_BedBack OR Entity_IO.RightPannel_BedBack OR CTBOX_RS232.CTBOX_KEY_BedBack), Q=> ); //获取上升沿
			F_TRIG_Jog(CLK:= (Entity_IO.LeftPannel_BedFore OR Entity_IO.RightPannel_BedFore OR CTBOX_RS232.CTBOX_KEY_BedFore)
						OR (Entity_IO.LeftPannel_BedBack OR Entity_IO.RightPannel_BedBack OR CTBOX_RS232.CTBOX_KEY_BedBack), Q=> ); //获取上升沿
	
			(*2.2.2 点动最大最小位置，绝对运动走记录值*)
			IF Entity_IO.LeftPannel_BedFore OR Entity_IO.RightPannel_BedFore OR CTBOX_RS232.CTBOX_KEY_BedFore THEN
				Axis_QJ.QJ_AxisCmd.AxisPara.rAbsPosition:=900;
			ELSE
				IF Entity_IO.LeftPannel_BedBack OR Entity_IO.RightPannel_BedBack OR CTBOX_RS232.CTBOX_KEY_BedBack THEN
					Axis_QJ.QJ_AxisCmd.AxisPara.rAbsPosition:=0;
				ELSE
					Axis_QJ.QJ_AxisCmd.AxisPara.rAbsPosition:=LIMIT(0,GVL_Retain.rBedRecordLength,900); 
				END_IF
			END_IF
			
			(*2.2.3 触发绝对运动，按键或者触发走记录位置*)
			Axis_QJ.QJ_AxisCmd.bAbs	:=R_TRIG_Jog.Q OR  Entity_IO.LeftPannel_MoveRecordPos OR Entity_IO.RightPannel_MoveRecordPos;
			
			(*2.2.4 触发停止*)
			R_RelStop(CLK:= (Axis_QJ.QJ_AxisState.rActPosition>901), Q=> ); 
			Axis_QJ.QJ_AxisCmd.bStop:=F_TRIG_Jog.Q OR R_RelStop.Q;
			
			IF Entity_IO.bXrayOneInput OR Entity_IO.bXayExpoInput OR Entity_IO.bXrayFluInput THEN 	//一档信号，或脚咋信号
				Step_StaticDR:=30;
			END_IF
	*)
END_ACTION

ACTION _a_QuickCT_entry:




Step_QuickCT:=0; 
GVL_State.iPLC_State:=240;
END_ACTION

ACTION _a_StandardCT_entry:

Step_StandardCT:=0; 

GVL_State.iPLC_State:=210;
END_ACTION

ACTION _a_StaticCT_exit:



	LampCmd5:=E_LampCmd.关闭;
	LampCmd6:=E_LampCmd.关闭;
	LampCmd7:=E_LampCmd.关闭;
	LampCmd8:=E_LampCmd.关闭;
	

	
	Entity_IO.bTriggerOut:=FALSE;
END_ACTION

ACTION _a_SystemInfo_active:

	LS_GetIPAddress_1(
		xExecute:= bGetPLC_IP, 
		eNetPort:= 0, 
		xDone=> , 
		xError=> , 
		diErrorID=> , 
		byIpSegmengt1=> , 
		byIpSegmengt2=> , 
		byIpSegmengt3=> , 
		byIpSegmengt4=> );
	
	LS_SetIPAddress_1(
		xExecute:= bSetPLC_IP, 
		eNetPort:= 0, 
		byIpSegmengt1:= , 
		byIpSegmengt2:= , 
		byIpSegmengt3:= , 
		byIpSegmengt4:= , 
		xDone=> , 
		xError=> , 
		diErrorID=> );
	
	GetPLCLoad(xEnable:= TRUE, xValid=> , xError=> , diErrorID=> , fLoad=> rPLC_Load);
	
	LS_SetDintDT_1(
		xExecute:= bSetSysTime, 
		uiYear:= , 
		uiMonth:= , 
		uiDay:= , 
		uiHour:= , 
		uiMinute:= , 
		uiSecond:= , 
		xDone=> , 
		xError=> , 
		diErrorID=> );

	LS_ReadDintDT_1(
		xEnable:= TRUE, 
		xValid=> , 
		xError=> , 
		diErrorID=> , 
		uiYear=> , 
		uiMonth=> , 
		uiDay=> , 
		uiHour=> , 
		uiMinute=> , 
		uiSecond=> );
END_ACTION

ACTION _a_HighDefinCT_entry:

Step_CBCT:=0; 
GVL_State.iPLC_State:=230;

Entity_io.bXraySwitch:=TRUE;//PF CLK信号切换继电器 不得电是默认BUCKY触发
END_ACTION

ACTION _a_Debug_active:


Entity_io.bTriggerOut:=aaa;

(*
Entity_IO.bXaryOne:=bbb;		//开启一档
Entity_IO.bXaryTwo:=ccc;		//开启二档
(**)

IF Entity_IO.bXrayOneInput THEN
	Entity_IO.bXaryOne:=TRUE;
ELSE
	Entity_IO.bXaryOne:=FALSE;
END_IF


IF Entity_IO.bXrayTwoInput THEN
	Entity_IO.bXaryTwo:=TRUE;
ELSE
	Entity_IO.bXaryTwo:=FALSE;
END_IF*)

(*
IF bTestFLU THEN
	Entity_IO.bXaryFlu:=TRUE;
ELSE
	Entity_IO.bXaryFlu:=FALSE;
END_IF
*)



IF bbb THEN
	Entity_IO.bXaryOne:=TRUE;
ELSE
	Entity_IO.bXaryOne:=FALSE;
END_IF


IF ccc THEN
	Entity_IO.bXaryTwo:=TRUE;
ELSE
	Entity_IO.bXaryTwo:=FALSE;
END_IF
END_ACTION

TRANSITION T_DR:

WorkStation_TCP.PLC_RECV1.m_nSocketType=1 AND (WorkStation_TCP.PLC_RECV1.m_nExpId=1 OR WorkStation_TCP.PLC_RECV1.m_nExpId=2)
END_TRANSITION

ACTION _a_DynamicsDR_entry:

Step_DynamicDR:=0;
GVL_State.iPLC_State:=120;
END_ACTION

ACTION _a_Homing_exit:


	Axis_XZ.XZ_AxisCmd.bHome:=FALSE;
	Axis_QJ.QJ_AxisCmd.bHome:=FALSE;
END_ACTION

ACTION _a_QuickCT_active:

	CASE Step_QuickCT OF 
		0:	//初始化准备流程
			(*1.给上位机发送的数据*)
			WorkStation_TCP.PLC_SEND1.m_nMoveState:=0;			//send[9] //0-准备过程中 1-准备完成 2-曝光中 3-本次扫描结束 
			bQuickCTLast		:=FALSE;
			bSendQuickCTAngle	:=FALSE;
			
			(*2.运动准备数据*)
			(*2.1 写入旋转速度参数*)
			IF WorkStation_TCP.PLC_RECV1.m_fSecondPerCicle<>0 THEN//避免除零
				Axis_XZ.XZ_AxisCmd.AxisPara.rAbsVelocity:=(LIMIT(360/300 ,360/WorkStation_TCP.PLC_RECV1.m_fSecondPerCicle ,360/8));
				XZ_Velocity:=LIMIT(360/300 ,360/(WorkStation_TCP.PLC_RECV1.m_fSecondPerCicle) ,360/8);
			ELSE
				Axis_XZ.XZ_AxisCmd.AxisPara.rAbsVelocity:=8;
			END_IF;
			
			(*3.中间变量复位*)
			FOR i:=1 TO 50 BY 1 DO 
				TON_CT_G[i](IN:= FALSE);
			END_FOR
			Axis_XZ.XZ_AxisCmd.bAbs		:=FALSE;
			Axis_QJ.QJ_AxisCmd.bAbs		:=FALSE;
			Step_QuickCT:=10;
				
		10://按5键，移动床到预设位置，松开即停，机架直接到预设位置
			(*1.发送给上位机的数据*)
			WorkStation_TCP.PLC_SEND1.m_nExpStates	:=1;		//0-准备过程中 1-准备完成 2-曝光中 3-本次扫描结束	
			WorkStation_TCP.PLC_SEND1.m_nMoveState	:=0;		//起始、终止状态， 默认值0， 1为当前扫描方案处于准备好状态，可以准备扫描；2为当前扫描方案结束，运动过程中值为0
			WorkStation_TCP.PLC_SEND1.m_nScanProType:=2;		//扫描方案类型 , 1-手动，0-自动. 
			
			(*2.旋转轴直接运动到目标位置*)
			Axis_XZ.XZ_AxisCmd.AxisPara.rAbsPosition	:=LIMIT(-3,WorkStation_TCP.PLC_RECV1.m_nRotateBegin,363);
			Axis_XZ.XZ_AxisCmd.AxisPara.rAbsVelocity	:=36;
			TON_CT_G[1](IN:=TRUE , PT:=T#500MS);
			Axis_XZ.XZ_AxisCmd.bAbs						:=TON_CT_G[1].Q;
			
			(*3.前进轴运动*)
			R_TRIG_G1(CLK:= CTBOX_RS232.CTBOX_KEY_MoveDistance, Q=> );//触发运动
			F_TRIG_G1(CLK:= CTBOX_RS232.CTBOX_KEY_MoveDistance, Q=> );//触发停止
			
			Axis_QJ.QJ_AxisCmd.bAbs	:=R_TRIG_G1.Q;
			Axis_QJ.QJ_AxisCmd.AxisPara.rAbsPosition	:=LIMIT(0,WorkStation_TCP.PLC_RECV1.m_fScanTop,900);
			Axis_QJ.QJ_AxisCmd.bStop:=F_TRIG_G1.Q;
			
			(*4.5灯逻辑处理*)
			IF ABS(Axis_QJ.QJ_AxisState.rActPosition-WorkStation_TCP.PLC_RECV1.m_fScanTop)>=1 THEN
				LampCmd5:=E_LampCmd.慢闪;
				WorkStation_TCP.PLC_SEND1.m_nFocus:=5;			//按键提示0228
			ELSE
				LampCmd5:=E_LampCmd.关闭;
				WorkStation_TCP.PLC_SEND1.m_nFocus:=0;			//关闭按键提示0228
			END_IF
			
			(*5.跳转*)
			TON_CT_G[2](IN:=ABS(Axis_QJ.QJ_AxisState.rActPosition-WorkStation_TCP.PLC_RECV1.m_fScanTop)<1 
				AND ABS(Axis_XZ.XZ_AxisState.rActPosition-WorkStation_TCP.PLC_RECV1.m_nRotateBegin)<1 
				AND Axis_XZ.XZ_AxisState.bStandStill AND Axis_QJ.QJ_AxisState.bStandStill, PT:=T#300MS);
			IF TON_CT_G[2].Q THEN  
				Step_QuickCT:=20;
			END_IF
			
		20:	//射线源参数写入成功标志
			(*1.变量复位*)
			LampCmd5:=E_LampCmd.关闭;
			Axis_XZ.XZ_AxisCmd.bAbs		:=FALSE;
			Axis_QJ.QJ_AxisCmd.bAbs		:=FALSE;
			Axis_QJ.QJ_AxisCmd.bStop	:=FALSE;
			
			(*2.射线源参数写入正常完毕*)
			IF DT_Xray.ExpPara_Step=66 THEN
				Step_QuickCT:=30;
			END_IF
			
		30:	//7灯和8灯开始慢闪
			(*1.给上位机发送的数*)
			WorkStation_TCP.PLC_SEND1.m_nMoveState	:=1;		//起始、终止状态， 默认值0， 1为当前扫描方案处于准备好状态
			WorkStation_TCP.PLC_SEND1.m_nFocus		:=8;		//按键提示0228
			
			(*2.CTBOX灯的状态*)
			LampCmd7:=E_LampCmd.慢闪;
			LampCmd8:=E_LampCmd.慢闪;
			
			TON_CT_G[3](IN:=TRUE , PT:=T#600MS);
			IF TON_CT_G[3].Q THEN
				Step_QuickCT:=40;
			END_IF
		
		40://用户选择自动扫描或手动扫描
			IF CTBOX_RS232.CTBOX_KEY_Auto=FALSE AND CTBOX_RS232.CTBOX_KEY_Manual THEN
				WorkStation_TCP.PLC_SEND1.m_nScanProType:=1;								//扫描方案类型 , 1-手动，0-自动. 
				bCBCT_AUTO_Manual:=TRUE;
			ELSIF CTBOX_RS232.CTBOX_KEY_Auto AND CTBOX_RS232.CTBOX_KEY_Manual=FALSE THEN
				WorkStation_TCP.PLC_SEND1.m_nScanProType:=0;								//扫描方案类型 , 1-手动，0-自动. 
				bCBCT_AUTO_Manual:=FALSE;
			ELSIF CTBOX_RS232.CTBOX_KEY_Auto=FALSE AND CTBOX_RS232.CTBOX_KEY_Manual=FALSE THEN
				;
			ELSIF CTBOX_RS232.CTBOX_KEY_Auto AND CTBOX_RS232.CTBOX_KEY_Manual THEN
				;
			END_IF
			
			IF (CTBOX_RS232.CTBOX_KEY_Auto AND CTBOX_RS232.CTBOX_KEY_Manual=FALSE) OR CTBOX_RS232.CTBOX_KEY_Manual AND CTBOX_RS232.CTBOX_KEY_Auto=FALSE THEN
				Step_QuickCT:=50;
			END_IF
			
		50://7和8灯关闭 
			(*1.给上位机发送的数据*)
			WorkStation_TCP.PLC_SEND1.m_nFocus:=0;	//关闭按键提示0228
			
			(*2.CTBOX灯关闭*)
			LampCmd7:=E_LampCmd.关闭;
			LampCmd8:=E_LampCmd.关闭;
			
			(*3.获取当前编码器数值*)
			iStartTrigger1:=Entity_IO.iEncoderPulse;//只赋值一次
			
			(*4.跳转*)
			TON_CT_G[4](IN:= TRUE, PT:=T#1S);
			IF TON_CT_G[4].Q THEN
				Step_QuickCT:=60;
			END_IF
			
		60://扫描中间态，给跳转用的
			(*1.变量复位*)
			FOR i:=1 TO 50 BY 1 DO 
				TON_CT_G[i](IN:= FALSE);
			END_FOR
			Axis_QJ.QJ_AxisCmd.bAbs:=FALSE;//复位前进轴
			Axis_XZ.XZ_AxisCmd.bAbs:=FALSE;//复位旋转轴
			iActNumPulse:=0;bSendQuickCTAngle:=FALSE;
			Step_QuickCT:=70;
			
		65://增加上位机扫描方案延迟
			DelayTime:=T#1MS*WorkStation_TCP.PLC_RECV1.m_nDelayTime;
			ExpTimeQuick:=T#1MS*REAL_TO_UDINT(WorkStation_TCP.PLC_RECV1.m_nMS);
			TON_CT_G[17](IN:=TRUE , PT:=DelayTime , Q=> , ET=> );
			IF TON_CT_G[17].Q THEN
				Step_QuickCT:=60;
			END_IF
			
		70:
			(*1.发送给上位机的数据*)
			WorkStation_TCP.PLC_SEND1.m_nExpStates	:=1;	//曝光状态
			WorkStation_TCP.PLC_SEND1.m_nMoveState	:=1;	//send[9]
			WorkStation_TCP.PLC_SEND1.m_nScanProType:=2;	//send[16]
			
			(*2.开启一二档信号*)
			Entity_IO.bXaryOne:=TRUE;//开启一二档
			Entity_IO.bXaryTwo:=TRUE;//开启一二档
			
			(*3.判断是否最后一次扫描*)
			IF WorkStation_TCP.PLC_RECV1.m_nLastMsg=1 THEN
				bQuickCTLast := TRUE;
			ELSE
				bQuickCTLast := FALSE;
			END_IF

			(*6.跳转指令*)
			TON_CT_G[5](IN:=TRUE,PT:=T#800MS);
			IF TON_CT_G[5].Q AND Entity_IO.bXaryOne AND Entity_IO.bXaryTwo THEN
				Step_QuickCT:=71;
			END_IF
			
		71://给增益校正预留的2档后2秒出束时间，此时旋转轴不运动
			TON_CT_G[13](IN:=TRUE,PT:=T#800MS);
			TON_CT_G[7](IN:=FALSE);
			IF Entity_IO.bXrayExp THEN
				WorkStation_TCP.PLC_SEND1.m_nExpStates	:=2;//
			END_IF;
			IF TON_CT_G[13].Q THEN
				Step_QuickCT:=80;
			END_IF
			
		74:
			Entity_IO.bXaryOne:=FALSE;
			Entity_IO.bXaryTwo:=FALSE;
			GVL_SCAN.bJumpScan:=TRUE;		//结束扫描，射线源超时报警了，EL019，结束扫描
			Step_QuickCT:=74;
			
		80://第一次自动扫描
			TON_CT_G[13](IN:=FALSE,PT:=T#2S);
			TON_CT_G[18](IN:=FALSE);
			(*1.给上位机发送的数*)
			IF Entity_IO.bXrayExp THEN
				WorkStation_TCP.PLC_SEND1.m_nExpStates	:=2;//
			END_IF;
			
			WorkStation_TCP.PLC_SEND1.m_nScanProType:=2;

			(*2.触发旋转轴运动*)
			Axis_XZ.XZ_AxisCmd.AxisPara.rAbsPosition:=LIMIT(-3,WorkStation_TCP.PLC_RECV1.m_nRotateEnd,363);
			Axis_XZ.XZ_AxisCmd.AxisPara.rAbsVelocity:=XZ_Velocity;
			TON_CT_G[6](IN:=TRUE , PT:=T#500MS );
			Axis_XZ.XZ_AxisCmd.bAbs:=TON_CT_G[6].Q;
			
			(*3.到达曝光角度后告诉上位机一声*)
			IF WorkStation_TCP.PLC_RECV1.m_nAngleStart<=WorkStation_TCP.PLC_RECV1.m_nAngleEnd THEN
				iAngleStartQuickCT:=WorkStation_TCP.PLC_RECV1.m_nAngleStart-0.2;
			ELSE
				iAngleStartQuickCT:=WorkStation_TCP.PLC_RECV1.m_nAngleStart+0.2;
			END_IF
			
			IF ABS(Axis_XZ.XZ_AxisState.rActPosition-iAngleStartQuickCT)<=0.2 THEN
				bSendQuickCTAngle:=TRUE;
			ELSE
				bSendQuickCTAngle:=FALSE;
			END_IF

			(*5.跳转,到达终止角度*)
			TON_CT_G[7](IN:= ABS(Axis_XZ.XZ_AxisState.rActPosition-WorkStation_TCP.PLC_RECV1.m_nRotateEnd)<1 AND Axis_XZ.XZ_AxisState.bStandStill, PT:=T#1S , Q=> , ET=> );	//100ms
			IF TON_CT_G[7].Q AND Entity_IO.bXrayExp=FALSE THEN
				Step_QuickCT:=85;
			END_IF
			
			(*6.一二档信号超时报警，射线源30秒连续开启曝光会报警*)
			TON_CT_G[8](IN:=Entity_IO.bXaryTwo , PT:=T#30S , Q=> , ET=> );
			IF TON_CT_G[8].Q THEN
				Step_QuickCT:=74;	
			END_IF
			
		85://解决处理bXrayExp变量有误差的问题
			bSendQuickCTAngle:=FALSE;
			TON_CT_G[18](IN:=TRUE , PT:=T#300MS , Q=> , ET=> );
			IF TON_CT_G[18].Q THEN
				Step_QuickCT:=90;
			END_IF
			
		90://出射线状态结束，采集射线源状态机信息
			(*1.关闭透视信号*)
			Entity_IO.bXaryOne		:=FALSE;
			Entity_IO.bXaryTwo		:=FALSE;
			Axis_XZ.XZ_AxisCmd.bAbs	:=FALSE;
			
			(*2.跳转*)
			IF GVL_State.iXray_State=40 OR DT_Xray.RadExp_Step=77 THEN	//DT射线源增加状态 ,回到待机状态 
				Step_QuickCT:=100;
			END_IF
			
		100://中间变量清零1070
			(*1.给上位机发送的数据*)
			WorkStation_TCP.PLC_SEND1.m_nExpStates	:=3;//结束
			WorkStation_TCP.PLC_SEND1.m_nMoveState	:=3;
			
			(*2.判断是否最后一次扫描*)
			TON_CT_G[9](IN:=TRUE , PT:=T#500MS , Q=> , ET=> );
			IF TON_CT_G[9].Q THEN
				IF (WorkStation_TCP.PLC_RECV1.m_nCircleIndex+1)>=(WorkStation_TCP.PLC_RECV1.m_nCircleCount) AND bQuickCTLast THEN//
					GVL_SCAN.bJumpScan:=TRUE;
				END_IF
			END_IF
			
			(*3.不是最后一次增加跳转判断增加跳转接着扫*)
			IF WorkStation_TCP.PLC_RECV1.m_nSocketType=1 THEN 	//增加第二次运动判断，m_nSocketType=1 
				Step_QuickCT:=105;
			END_IF
		
		105://多次扫再次写入射线源参数，保证成功
			IF DT_Xray.ExpPara_Step=66 THEN
				Step_QuickCT:=110;
			END_IF
		
		110://CBCT下的自动扫还是手动扫，根据上位机命令
			IF WorkStation_TCP.PLC_RECV1.m_nScanMoveType=1 THEN
				Step_QuickCT:=200;		//手动扫描
			ELSE
				Step_QuickCT:=120;		//自动扫描
			END_IF
		 
		120://开启自动扫描
			(*1.前进轴自动运动*)
			TON_CT_G[10](IN:=TRUE , PT:=T#300MS , Q=> , ET=> );
			Axis_QJ.QJ_AxisCmd.AxisPara.rAbsPosition:=LIMIT(0,WorkStation_TCP.PLC_RECV1.m_fScanTop,900);
			Axis_QJ.QJ_AxisCmd.bAbs:=TON_CT_G[10].Q;
			
			(*2.给上位机发送的数据*)
			IF ABS(Axis_QJ.QJ_AxisState.rActPosition-WorkStation_TCP.PLC_RECV1.m_fScanTop)<1 AND Axis_QJ.QJ_AxisState.bStandStill THEN
				WorkStation_TCP.PLC_SEND1.m_nMoveState:=1; 			//send [9]
				Step_QuickCT:=60;				//自动扫描
			ELSE
				WorkStation_TCP.PLC_SEND1.m_nMoveState:=0; 			//send [9]	//0-准备过程中 1-准备完成 2-曝光中 3-本次扫描结束
			END_IF
			
		(*-------------------------手动扫描-----------------------------*)	
		200://中间状态清零
			WorkStation_TCP.PLC_SEND1.m_nMoveState:=0; //send [9]	//0-准备过程中 1-准备完成 2-曝光中 3-本次扫描结束
			Axis_XZ.XZ_AxisCmd.bAbs:=FALSE;
			Step_QuickCT:=210;
			
		210://7灯闪烁，机架运动到目标位置
			(*1.发送给上位机的数据*)
			WorkStation_TCP.PLC_SEND1.m_nMoveState:=0; //send [9]	//0-准备过程中 1-准备完成 2-曝光中 3-本次扫描结束
			
			(*2.7灯闪烁*)
			LampCmd7:=E_LampCmd.慢闪;
			WorkStation_TCP.PLC_SEND1.m_nFocus:=7;	//按键提示0228
			
			(*3.旋转轴运动到目标位置*)
			Axis_XZ.XZ_AxisCmd.AxisPara.rAbsPosition:=LIMIT(-4,WorkStation_TCP.PLC_RECV1.m_nRotateBegin,363);
			Axis_XZ.XZ_AxisCmd.AxisPara.rAbsVelocity:=XZ_Velocity;
			
			IF WorkStation_TCP.PLC_RECV1.m_nSocketType=1 THEN
				Axis_XZ.XZ_AxisCmd.bAbs:=TRUE;
			END_IF;
			
			(*4.到位后2秒跳转*)
			IF ABS(Axis_XZ.XZ_AxisState.rActPosition-WorkStation_TCP.PLC_RECV1.m_nRotateBegin)<1 AND Axis_XZ.XZ_AxisState.bStandStill THEN
				Step_QuickCT:=220;
			END_IF
		
		220://中间状态清零
			Axis_XZ.XZ_AxisCmd.bAbs:=FALSE;
			Axis_QJ.QJ_AxisCmd.bAbs:=FALSE;
			Step_QuickCT:=230;
			
		230://用户按7键，床自动走到预设位置
			(*1.按7键关闭7灯*)
			IF CTBOX_RS232.CTBOX_KEY_Manual THEN
				LampCmd7:=E_LampCmd.关闭;
				WorkStation_TCP.PLC_SEND1.m_nFocus:=0;	//关闭按键提示0228
			END_IF
			
			(*2.触发床运动*)
			R_TRIG_G2(CLK:=CTBOX_RS232.CTBOX_KEY_Manual , Q=> );
			Axis_QJ.QJ_AxisCmd.AxisPara.rAbsPosition:=LIMIT(0,WorkStation_TCP.PLC_RECV1.m_fScanTop,900);
			Axis_QJ.QJ_AxisCmd.bAbs:=R_TRIG_G2.Q;
			
			(*3.跳转指令*)
			IF ABS(Axis_QJ.QJ_AxisState.rActPosition-WorkStation_TCP.PLC_RECV1.m_fScanTop)<1 AND (LampCmd7=E_LampCmd.关闭) THEN //保证必须按下7键
				WorkStation_TCP.PLC_SEND1.m_nMoveState:=1; //send [9]	//0-准备过程中 1-准备完成 2-曝光中 3-本次扫描结束
			ELSE
				WorkStation_TCP.PLC_SEND1.m_nMoveState:=0; //send [9]	//0-准备过程中 1-准备完成 2-曝光中 3-本次扫描结束
			END_IF
			
			(*4.延迟跳转，保证send [9]发送*)
			TON_CT_G[11](IN:=(WorkStation_TCP.PLC_SEND1.m_nMoveState=1) , PT:=T#1100MS , Q=> , ET=> );
			IF TON_CT_G[11].Q THEN
				Step_QuickCT:=60;
			END_IF
	END_CASE
END_ACTION

ACTION _a_MovePos_active:

END_ACTION

ACTION _a_StandardCT_exit:


	LampCmd5:=E_LampCmd.关闭;
	LampCmd6:=E_LampCmd.关闭;
	LampCmd7:=E_LampCmd.关闭;
	LampCmd8:=E_LampCmd.关闭;
	

	Entity_IO.bTriggerOut:=FALSE;
END_ACTION

TRANSITION T_StaticCT:


(*进入定位片扫描*)
	WorkStation_TCP.PLC_RECV1.m_nSocketType=1 AND WorkStation_TCP.PLC_RECV1.m_nExpId=4
END_TRANSITION

ACTION _a_StaticDR_entry:



Step_StaticDR:=0; 
bXrayOneDR:=FALSE;
Entity_IO.bXaryTwo:=FALSE;Entity_IO.bXaryOne:=FALSE;
GVL_State.iPLC_State:=110;
TOF_DR111(IN:=FALSE);TOF_DR22(IN:=FALSE);
END_ACTION

ACTION AirHigh_active:

	CASE Step_Air OF 
	
		0://高清校正  透视模式
			(*1.给上位机发送的数据*)
			WorkStation_TCP.PLC_SEND1.m_nMoveState:=0;			//send[9] //0-准备过程中 1-准备完成 2-曝光中 3-本次扫描结束 
			bAirLast2		:=FALSE;
			Entity_IO.bXraySwitch:=TRUE;//透视触发
			(*2.中间变量复位*)
			FOR i:=1 TO 50 BY 1 DO 
				TON_Air[i](IN:= FALSE);
			END_FOR
			Axis_XZ.XZ_AxisCmd.bAbs		:=FALSE;
			Axis_QJ.QJ_AxisCmd.bAbs		:=FALSE;
			iTriggerNum2:=0;
			bAirHigh:=FALSE;
			Entity_IO.bXaryFlu:=FALSE;	//开启透视模式
			Step_Air:=10;
			
		10:
			(*1.发送给上位机的数据*)
			WorkStation_TCP.PLC_SEND1.m_nExpStates	:=1;		//0-准备过程中 1-准备完成 2-曝光中 3-本次扫描结束	
			WorkStation_TCP.PLC_SEND1.m_nMoveState	:=0;		//起始、终止状态， 默认值0， 1为当前扫描方案处于准备好状态，可以准备扫描；2为当前扫描方案结束，运动过程中值为0
			WorkStation_TCP.PLC_SEND1.m_nScanProType:=2;		//扫描方案类型 , 1-手动，0-自动. 
		
			(*2.旋转轴和前进轴自动运动到目标位置*)
			(*2.1 旋转轴直接运动到目标位置*)
			Axis_XZ.XZ_AxisCmd.AxisPara.rAbsPosition	:=MIN(LIMIT(-3,WorkStation_TCP.PLC_RECV1.m_nRotateBegin,363),LIMIT(-3,WorkStation_TCP.PLC_RECV1.m_nRotateEnd,363));
			Axis_XZ.XZ_AxisCmd.AxisPara.rAbsVelocity	:=30;
			TON_Air[21](IN:=TRUE , PT:=T#500MS);
			Axis_XZ.XZ_AxisCmd.bAbs						:=TON_Air[21].Q;

			(*2.2 前进轴直接运动到目标位置*)
			Axis_QJ.QJ_AxisCmd.AxisPara.rAbsPosition	:=LIMIT(0,WorkStation_TCP.PLC_RECV1.m_fScanTop,900);
			Axis_QJ.QJ_AxisCmd.AxisPara.rAbsVelocity	:=60;
			TON_Air[22](IN:=TRUE , PT:=T#500MS);
			Axis_QJ.QJ_AxisCmd.bAbs						:=TON_Air[22].Q;
			
			(*5.跳转*)
			TON_Air[23](IN:=ABS(Axis_QJ.QJ_AxisState.rActPosition-WorkStation_TCP.PLC_RECV1.m_fScanTop)<1 
				AND ABS(Axis_XZ.XZ_AxisState.rActPosition-MIN(WorkStation_TCP.PLC_RECV1.m_nRotateBegin,WorkStation_TCP.PLC_RECV1.m_nRotateEnd))<1 
				AND Axis_XZ.XZ_AxisState.bStandStill AND Axis_QJ.QJ_AxisState.bStandStill, PT:=T#150MS);
			IF TON_Air[23].Q AND DT_Xray.FluPara_Setp=66 THEN  //机架运动到目标位置，并且射线源参数写入成功
				Step_Air:=20;
			END_IF
			
		20:
			//8灯开始慢闪
			(*1.给上位机发送的数*)
			WorkStation_TCP.PLC_SEND1.m_nMoveState	:=1;		//起始、终止状态， 默认值0， 1为当前扫描方案处于准备好状态
			WorkStation_TCP.PLC_SEND1.m_nFocus		:=8;		//按键提示0228
			
			(*2.CTBOX灯的状态*)
			LampCmd8:=E_LampCmd.慢闪;
			
			(*3.跳转*)
			TON_Air[1](IN:=TRUE , PT:=T#600MS);
			IF TON_Air[1].Q THEN
				Step_Air:=30;
			END_IF
			
		30:
			IF CTBOX_RS232.CTBOX_KEY_Auto THEN //按8键
				bAirHigh:=TRUE;
				LampCmd8:=E_LampCmd.关闭;
			END_IF
			
			TON_Air[2](IN:=bAirHigh , PT:=T#600MS);
			IF TON_Air[2].Q THEN
				Step_Air:=40;
			END_IF
		40:
			(*1.给上位机发送的数据*)
			WorkStation_TCP.PLC_SEND1.m_nMoveState:=0;			//send[9] //0-准备过程中 1-准备完成 2-曝光中 3-本次扫描结束 
			bAirLast2		:=FALSE;
			(*2.中间变量复位*)
			FOR i:=1 TO 50 BY 1 DO 
				TON_Air[i](IN:= FALSE);
			END_FOR
			iTriggerNum2:=0;
			Entity_IO.bXaryFlu:=FALSE;	//开启透视模式
			Step_Air:=45;
			
		45:
			TON_Air[3](IN:=TRUE , PT:=T#8S);
			IF TON_Air[3].Q THEN
				Step_Air:=46;
			END_IF
			
		46:
			FOR i:=1 TO 50 BY 1 DO 
				TON_Air[i](IN:= FALSE);
			END_FOR
			Step_Air:=50;
			
		50://开启透视模式
			(*1.发送给上位机的数据*)
			WorkStation_TCP.PLC_SEND1.m_nMoveState	:=1;	//send[9]
			WorkStation_TCP.PLC_SEND1.m_nScanProType:=2;	//send[16]
			
			(*2.射线源参数写入成功，开启透视*)
			IF DT_Xray.FluPara_Setp=66 THEN  //保证写入参数
				Entity_IO.bXaryFlu:=TRUE;//开启透视模式
			END_IF;
			
			(*3.判断是否最后一次扫描*)
			IF WorkStation_TCP.PLC_RECV1.m_nLastMsg=1 THEN
				bAirLast2 := TRUE;
			ELSE
				bAirLast2 := FALSE;
			END_IF
			
			F_Trig_Air2(CLK:= FALSE, Q=> );
			
			(*4.跳转指令*)
			TON_Air[24](IN:=TRUE,PT:=T#1S);
			IF TON_Air[24].Q AND Entity_IO.bXaryFlu THEN
				Step_Air:=60;
			END_IF
			iTriggerNum2:=0;
			
		60:
			(*1.发送给上位机的数据*)
			WorkStation_TCP.PLC_SEND1.m_nMoveState	:=2;			//send[9]//0-准备过程中 1-准备完成 2-曝光中 3-本次扫描结束	
			WorkStation_TCP.PLC_SEND1.m_nScanProType:=2;			//send[16]
			
			(*2.触发四次采集图像*)
			Blink_Air2(ENABLE:= TRUE, TIMELOW:= T#50MS, TIMEHIGH:=T#10MS , OUT=> );
			IF iTriggerNum2<50 THEN
				Entity_IO.bTriggerOut:=Blink_Air2.OUT;
				F_Trig_Air2(CLK:= Entity_IO.bTriggerOut, Q=> );
			ELSE
				F_Trig_Air2(CLK:= FALSE);
				Entity_IO.bTriggerOut:=FALSE;
			END_IF;
			
			(*3.计数触发了几次几个脉冲*)
			IF F_Trig_Air2.Q THEN
				iTriggerNum2:=iTriggerNum2+1;
			END_IF;
			
			(*4.曝光次数满足，跳出，EL069*)
			IF iTriggerNum2>=33 THEN
				Step_Air:=70;
			END_IF
	
		70:
			(*1.运动变量复位*)
			Entity_IO.bXaryFlu:=FALSE;
			Axis_QJ.QJ_AxisCmd.bAbs:=FALSE;
			Axis_XZ.XZ_AxisCmd.bAbs:=FALSE;	
			Entity_IO.bTriggerOut:=FALSE;

			(*2.给上位机发送数据，不能太快*)
			TON_Air[25](IN:=TRUE , PT:=T#3S , Q=> , ET=> );			//留些时间给上位机发送本次扫描结束方案标志
			
			(*2.扫描结束，发送结束标志位*)
			IF DT_Xray.RadFlu_Step=66 THEN 
				WorkStation_TCP.PLC_SEND1.m_nMoveState:=3;			//send[9] //0-准备过程中 1-准备完成 2-曝光中 3-本次扫描结束
			END_IF;
			
			(*3.判断师傅最后一次扫描*)
			IF TON_Air[25].Q THEN
				IF (WorkStation_TCP.PLC_RECV1.m_nCircleIndex+1)>=(WorkStation_TCP.PLC_RECV1.m_nCircleCount) AND bAirLast2 AND DT_Xray.RadFlu_Step=66 THEN 	//用于区分自动扫是否最后一次，此时=1，=1都等于1
					Step_Air:=300;
				END_IF;
			END_IF
			
			IF WorkStation_TCP.PLC_RECV1.m_nSocketType=1 AND WorkStation_TCP.PLC_RECV1.m_nExpId = 8 THEN
				Step_Air:=300;
			END_IF
			
			(*4.不是最后一次，收到下一次命令，继续扫*)
			IF WorkStation_TCP.PLC_RECV1.m_nSocketType=1 AND DT_Xray.RadFlu_Step=66 AND WorkStation_TCP.PLC_RECV1.m_nExpId = 7 THEN 	//增加第二次运动判断，m_nSocketType=1 
				Step_Air:=40;
			END_IF

			
		300://快速扫描校正
				//初始化准备流程
				(*1.给上位机发送的数据*)
				WorkStation_TCP.PLC_SEND1.m_nMoveState:=0;			//send[9] //0-准备过程中 1-准备完成 2-曝光中 3-本次扫描结束 
				bAirLast3		:=FALSE;
				Entity_IO.bXraySwitch:=FALSE;//
				(*2.中间变量复位*)
				FOR i:=1 TO 50 BY 1 DO 
					TON_Air[i](IN:= FALSE);
				END_FOR
				Axis_XZ.XZ_AxisCmd.bAbs		:=FALSE;
				Axis_QJ.QJ_AxisCmd.bAbs		:=FALSE;
				Step_Air:=310;
				
			310:
				(*1.发送给上位机的数据*)
				WorkStation_TCP.PLC_SEND1.m_nExpStates	:=1;		//0-准备过程中 1-准备完成 2-曝光中 3-本次扫描结束	
				WorkStation_TCP.PLC_SEND1.m_nMoveState	:=0;		//起始、终止状态， 默认值0， 1为当前扫描方案处于准备好状态，可以准备扫描；2为当前扫描方案结束，运动过程中值为0
				WorkStation_TCP.PLC_SEND1.m_nScanProType:=2;		//扫描方案类型 , 1-手动，0-自动. 
			
				(*2.旋转轴和前进轴自动运动到目标位置*)
				(*2.1 旋转轴直接运动到目标位置*)
				Axis_XZ.XZ_AxisCmd.AxisPara.rAbsPosition	:=LIMIT(-3,WorkStation_TCP.PLC_RECV1.m_nRotateBegin,363);
				Axis_XZ.XZ_AxisCmd.AxisPara.rAbsVelocity	:=30;
				TON_Air[31](IN:=TRUE , PT:=T#500MS);
				Axis_XZ.XZ_AxisCmd.bAbs						:=TON_Air[31].Q;
	
				(*2.2 前进轴直接运动到目标位置*)
				Axis_QJ.QJ_AxisCmd.AxisPara.rAbsPosition	:=LIMIT(0,WorkStation_TCP.PLC_RECV1.m_fScanTop,900);
				Axis_QJ.QJ_AxisCmd.AxisPara.rAbsVelocity	:=60;
				TON_Air[32](IN:=TRUE , PT:=T#500MS);
				Axis_QJ.QJ_AxisCmd.bAbs						:=TON_Air[32].Q;
				
				(*5.跳转*)
				TON_Air[33](IN:=ABS(Axis_QJ.QJ_AxisState.rActPosition-WorkStation_TCP.PLC_RECV1.m_fScanTop)<1 
					AND ABS(Axis_XZ.XZ_AxisState.rActPosition-WorkStation_TCP.PLC_RECV1.m_nRotateBegin)<1 
					AND Axis_XZ.XZ_AxisState.bStandStill AND Axis_QJ.QJ_AxisState.bStandStill, PT:=T#150MS);
				IF TON_Air[33].Q THEN  
					Step_Air:=320;
				END_IF
				
			320://写入射线源参数成功
				(*1.变量复位*)
				Axis_XZ.XZ_AxisCmd.bAbs		:=FALSE;
				Axis_QJ.QJ_AxisCmd.bAbs		:=FALSE;
				
				(*2.射线源参数写入正常完毕*)
				IF DT_Xray.ExpPara_Step=66 THEN
					Step_Air:=330;
				END_IF
				
			330:
				//扫描中间态，跳转使用
				(*1.变量复位*)
				FOR i:=1 TO 50 BY 1 DO 
					TON_Air[i](IN:= FALSE);
				END_FOR
				Axis_QJ.QJ_AxisCmd.bAbs:=FALSE;//复位前进轴
				Axis_XZ.XZ_AxisCmd.bAbs:=FALSE;//复位旋转轴
				Step_Air:=340;
				
			340://开启曝光
				(*1.发送给上位机的数据*)
				WorkStation_TCP.PLC_SEND1.m_nMoveState	:=1;	//send[9]
				WorkStation_TCP.PLC_SEND1.m_nScanProType:=2;	//send[16]
				
				(*2.射线源参数写入成功，开启透视*)
				IF DT_Xray.ExpPara_Step=66 THEN  //保证写入参数
					Entity_IO.bXaryOne:=TRUE;//开启一二档
					Entity_IO.bXaryTwo:=TRUE;//开启一二档
				END_IF;
				
				(*3.判断是否最后一次扫描*)
				IF WorkStation_TCP.PLC_RECV1.m_nLastMsg=1 THEN
					bAirLast3 := TRUE;
				ELSE
					bAirLast3 := FALSE;
				END_IF
				
				(*4.跳转指令*)
				TON_Air[34](IN:=TRUE,PT:=T#2S);//把曝光的时间加这这里了
				
				IF TON_Air[34].Q AND Entity_IO.bXaryOne AND Entity_IO.bXaryTwo THEN
					Step_Air:=350;
				END_IF
				
				IF Entity_IO.bXrayExp THEN
					WorkStation_TCP.PLC_SEND1.m_nExpStates	:=2;//
				END_IF;
				
			350:
				(*1.发送给上位机的数据*)
			//	WorkStation_TCP.PLC_SEND1.m_nMoveState	:=2;			//send[9]//0-准备过程中 1-准备完成 2-曝光中 3-本次扫描结束	
				(*1.给上位机发送的数*)
				IF Entity_IO.bXrayExp THEN
					WorkStation_TCP.PLC_SEND1.m_nExpStates	:=2;//
				END_IF;
				WorkStation_TCP.PLC_SEND1.m_nScanProType:=2;			//send[16]
				
				(*2.曝光结束，跳出*)
				IF DT_Xray.RadExp_Step=66 THEN
					Step_Air:=360;	
				END_IF
			
			360:
				(*1.运动变量复位*)
				Entity_IO.bXaryOne:=FALSE;
				Entity_IO.bXaryTwo:=FALSE;
				Axis_QJ.QJ_AxisCmd.bAbs:=FALSE;
				Axis_XZ.XZ_AxisCmd.bAbs:=FALSE;	
				Entity_IO.bTriggerOut:=FALSE;
	
				(*2.给上位机发送数据，不能太快*)
				TON_Air[36](IN:=TRUE , PT:=T#1600MS , Q=> , ET=> );	//留些时间给上位机发送本次扫描结束方案标志
				
				(*2.扫描结束，发送结束标志位*)
				IF DT_Xray.RadExp_Step=77 THEN 
					WorkStation_TCP.PLC_SEND1.m_nMoveState:=3;			//send[9] //0-准备过程中 1-准备完成 2-曝光中 3-本次扫描结束
				END_IF;
				
				(*3.判断师傅最后一次扫描*)
				IF TON_Air[36].Q THEN
					IF (WorkStation_TCP.PLC_RECV1.m_nCircleIndex+1)>=(WorkStation_TCP.PLC_RECV1.m_nCircleCount) AND bAirLast3 AND DT_Xray.RadExp_Step=77 THEN 	//用于区分自动扫是否最后一次，此时=1，=1都等于1
						GVL_SCAN.bJumpScan:=TRUE;
					END_IF;
				END_IF
				
				(*4.不是最后一次，收到下一次命令，继续扫*)
				IF WorkStation_TCP.PLC_RECV1.m_nSocketType=1 AND DT_Xray.RadExp_Step=77 THEN 	//增加第二次运动判断，m_nSocketType=1 
					Step_Air:=300;
				END_IF
	END_CASE
END_ACTION

TRANSITION T_AirCal:
(*进入空气校正/高清校正模式*)
	WorkStation_TCP.PLC_RECV1.m_nSocketType=1 AND (WorkStation_TCP.PLC_RECV1.m_nExpId=7  OR WorkStation_TCP.PLC_RECV1.m_nExpId=8)
END_TRANSITION

TRANSITION T_AirCal_Quick:
(*进入空气校正/快速校正模式*)
	WorkStation_TCP.PLC_RECV1.m_nSocketType=1 AND WorkStation_TCP.PLC_RECV1.m_nExpId=8
END_TRANSITION

ACTION _AirCalQuick_active:

